LIN {X 0,Y 210.319,Z 902.747,A -85,B 0,C 180,E1 -29716.885,E2 -29716.885} C_VEL
LIN {X 0,Y 210.36,Z 916.958,A -85,B 0,C 180,E1 -29720.636,E2 -29720.636} C_VEL
LIN {X 0,Y 210.916,Z 920.236,A -85,B 0,C 180,E1 -29721.95,E2 -29721.95} C_VEL
LIN {X 0,Y 215.207,Z 930.512,A -85,B 0,C 180,E1 -29727.206,E2 -29727.206} C_VEL
LIN {X 0,Y 222.813,Z 941.87,A -85,B 0,C 180,E1 -29733.503,E2 -29733.503} C_VEL
LIN {X 0,Y 234.173,Z 953.754,A -85,B 0,C 180,E1 -29740.198,E2 -29740.198} C_VEL
LIN {X 0,Y 249.698,Z 966.285,A -85,B 0,C 180,E1 -29747.036,E2 -29747.036} C_VEL
LIN {X 0,Y 259.021,Z 973.419,A -85,B 0,C 180,E1 -29750.555,E2 -29750.555} C_VEL
LIN {X 0,Y 266.825,Z 979.349,A -85,B 0,C 180,E1 -29753.45,E2 -29753.45} C_VEL
LIN {X 0,Y 272.417,Z 983.731,A -85,B 0,C 180,E1 -29755.644,E2 -29755.644} C_VEL
LIN {X 0,Y 279.791,Z 989.154,A -85,B 0,C 180,E1 -29758.652,E2 -29758.652} C_VEL
LIN {X 0,Y 286.884,Z 994.471,A -85,B 0,C 180,E1 -29761.873,E2 -29761.873} C_VEL
LIN {X 0,Y 291.933,Z 998.076,A -85,B 0,C 180,E1 -29764.322,E2 -29764.322} C_VEL
LIN {X 0,Y 297.29,Z 1001.982,A -85,B 0,C 180,E1 -29767.214,E2 -29767.214} C_VEL
LIN {X 0,Y 301.306,Z 1004.65,A -85,B 0,C 180,E1 -29769.521,E2 -29769.521} C_VEL
LIN {X 0,Y 304.104,Z 1006.607,A -85,B 0,C 180,E1 -29771.355,E2 -29771.355} C_VEL
LIN {X 0,Y 307.657,Z 1009.394,A -85,B 0,C 180,E1 -29774.091,E2 -29774.091} C_VEL
LIN {X 0,Y 310.964,Z 1011.661,A -85,B 0,C 180,E1 -29776.938,E2 -29776.938} C_VEL
LIN {X 0,Y 314.05,Z 1013.321,A -85,B 0,C 180,E1 -29779.947,E2 -29779.947} C_VEL
LIN {X 0,Y 316.064,Z 1014.25,A -85,B 0,C 180,E1 -29782.333,E2 -29782.333} C_VEL
LIN {X 0,Y 317.605,Z 1014.95,A -85,B 0,C 180,E1 -29784.922,E2 -29784.922} C_VEL
LIN {X 0,Y 318.555,Z 1015.361,A -85,B 0,C 180,E1 -29787.471,E2 -29787.471} C_VEL
LIN {X 0,Y 318.776,Z 1015.511,A -85,B 0,C 180,E1 -29790,E2 -29790} C_VEL
LIN {X 0,Y 318.553,Z 1015.357,A -85,B 0,C 180,E1 -29792.529,E2 -29792.529} C_VEL
LIN {X 0,Y 317.534,Z 1014.981,A -85,B 0,C 180,E1 -29795.143,E2 -29795.143} C_VEL
LIN {X 0,Y 316.037,Z 1014.273,A -85,B 0,C 180,E1 -29797.667,E2 -29797.667} C_VEL
LIN {X 0,Y 313.796,Z 1013.227,A -85,B 0,C 180,E1 -29800.321,E2 -29800.321} C_VEL
LIN {X 0,Y 310.634,Z 1011.462,A -85,B 0,C 180,E1 -29803.382,E2 -29803.382} C_VEL
LIN {X 0,Y 307.344,Z 1009.146,A -85,B 0,C 180,E1 -29806.179,E2 -29806.179} C_VEL
LIN {X 0,Y 303.767,Z 1006.331,A -85,B 0,C 180,E1 -29808.899,E2 -29808.899} C_VEL
LIN {X 0,Y 300.741,Z 1004.289,A -85,B 0,C 180,E1 -29810.813,E2 -29810.813} C_VEL
LIN {X 0,Y 295.368,Z 1000.609,A -85,B 0,C 180,E1 -29813.859,E2 -29813.859} C_VEL
LIN {X 0,Y 290.463,Z 996.916,A -85,B 0,C 180,E1 -29816.462,E2 -29816.462} C_VEL
LIN {X 0,Y 285.122,Z 993.212,A -85,B 0,C 180,E1 -29818.951,E2 -29818.951} C_VEL
LIN {X 0,Y 278.129,Z 987.907,A -85,B 0,C 180,E1 -29822.048,E2 -29822.048} C_VEL
LIN {X 0,Y 270.582,Z 982.305,A -85,B 0,C 180,E1 -29825.098,E2 -29825.098} C_VEL
LIN {X 0,Y 263.436,Z 976.696,A -85,B 0,C 180,E1 -29827.849,E2 -29827.849} C_VEL
LIN {X 0,Y 253.442,Z 969.085,A -85,B 0,C 180,E1 -29831.522,E2 -29831.522} C_VEL
LIN {X 0,Y 239.695,Z 958.548,A -85,B 0,C 180,E1 -29837.138,E2 -29837.138} C_VEL
LIN {X 0,Y 225.348,Z 945.049,A -85,B 0,C 180,E1 -29844.763,E2 -29844.763} C_VEL
LIN {X 0,Y 217.144,Z 933.823,A -85,B 0,C 180,E1 -29850.957,E2 -29850.957} C_VEL
LIN {X 0,Y 212.466,Z 924.491,A -85,B 0,C 180,E1 -29855.923,E2 -29855.923} C_VEL
LIN {X 0,Y 209.033,Z 913.185,A -85,B 0,C 180,E1 -29861.437,E2 -29861.437} C_VEL
LIN {X 0,Y 207.187,Z 900.869,A -85,B 0,C 180,E1 -29866.932,E2 -29866.932} C_VEL
LIN {X 0,Y 206.615,Z 891.892,A -85,B 0,C 180,E1 -29870.748,E2 -29870.748} C_VEL
LIN {X 0,Y 206.248,Z 887.985,A -85,B 0,C 180,E1 -29872.997,E2 -29872.997} C_VEL
LIN {X 0,Y 205.868,Z 884.919,A -85,B 0,C 180,E1 -29875.595,E2 -29875.595} C_VEL
LIN {X 0,Y 205.707,Z 883.432,A -85,B 0,C 180,E1 -29877.553,E2 -29877.553} C_VEL
LIN {X 0,Y 205.644,Z 882.867,A -85,B 0,C 180,E1 -29879.359,E2 -29879.359} C_VEL
LIN {X 0,Y 202.968,Z 897.04,A -85,B 0,C 180,E1 -29879.559,E2 -29879.559} C_VEL
LIN {X 0,Y 199.768,Z 909.589,A -85,B 0,C 180,E1 -29879.721,E2 -29879.721} C_VEL
LIN {X 0,Y 196.126,Z 921.044,A -85,B 0,C 180,E1 -29879.878,E2 -29879.878} C_VEL
LIN {X 0,Y 191.11,Z 933.924,A -85,B 0,C 180,E1 -29880.105,E2 -29880.105} C_VEL
LIN {X 0,Y 185.363,Z 946.249,A -85,B 0,C 180,E1 -29880.387,E2 -29880.387} C_VEL
LIN {X 0,Y 178.348,Z 958.97,A -85,B 0,C 180,E1 -29880.8,E2 -29880.8} C_VEL
LIN {X 0,Y 171.342,Z 969.953,A -85,B 0,C 180,E1 -29881.224,E2 -29881.224} C_VEL
LIN {X 0,Y 163.472,Z 980.735,A -85,B 0,C 180,E1 -29881.747,E2 -29881.747} C_VEL
LIN {X 0,Y 154.751,Z 991.222,A -85,B 0,C 180,E1 -29882.433,E2 -29882.433} C_VEL
LIN {X 0,Y 146.063,Z 1000.482,A -85,B 0,C 180,E1 -29883.257,E2 -29883.257} C_VEL
LIN {X 0,Y 135.659,Z 1010.198,A -85,B 0,C 180,E1 -29884.256,E2 -29884.256} C_VEL
LIN {X 0,Y 125.327,Z 1018.712,A -85,B 0,C 180,E1 -29885.529,E2 -29885.529} C_VEL
LIN {X 0,Y 113.37,Z 1027.307,A -85,B 0,C 180,E1 -29887.326,E2 -29887.326} C_VEL
LIN {X 0,Y 103.236,Z 1033.736,A -85,B 0,C 180,E1 -29889.215,E2 -29889.215} C_VEL
LIN {X 0,Y 89.923,Z 1040.997,A -85,B 0,C 180,E1 -29892.335,E2 -29892.335} C_VEL
LIN {X 0,Y 80.172,Z 1045.652,A -85,B 0,C 180,E1 -29895.365,E2 -29895.365} C_VEL
LIN {X 0,Y 67.643,Z 1050.762,A -85,B 0,C 180,E1 -29900.762,E2 -29900.762} C_VEL
LIN {X 0,Y 55.947,Z 1054.78,A -85,B 0,C 180,E1 -29908.441,E2 -29908.441} C_VEL
LIN {X 0,Y 49.911,Z 1056.686,A -85,B 0,C 180,E1 -29914.283,E2 -29914.283} C_VEL
LIN {X 0,Y 41.398,Z 1058.964,A -85,B 0,C 180,E1 -29927.23,E2 -29927.23} C_VEL
LIN {X 0,Y 35.44,Z 1060.469,A -85,B 0,C 180,E1 -29946.634,E2 -29946.634} C_VEL
LIN {X 0,Y 34.109,Z 1060.992,A -85,B 0,C 180,E1 -29970,E2 -29970} C_VEL
LIN {X 0,Y 35.44,Z 1060.469,A -85,B 0,C 180,E1 -29993.366,E2 -29993.366} C_VEL
LIN {X 0,Y 41.398,Z 1058.964,A -85,B 0,C 180,E1 -30012.769,E2 -30012.769} C_VEL
LIN {X 0,Y 50.596,Z 1056.467,A -85,B 0,C 180,E1 -30026.449,E2 -30026.449} C_VEL
LIN {X 0,Y 64.625,Z 1051.854,A -85,B 0,C 180,E1 -30037.571,E2 -30037.571} C_VEL
LIN {X 0,Y 73.824,Z 1048.354,A -85,B 0,C 180,E1 -30042.169,E2 -30042.169} C_VEL
LIN {X 0,Y 86.648,Z 1042.62,A -85,B 0,C 180,E1 -30046.729,E2 -30046.729} C_VEL
LIN {X 0,Y 96.543,Z 1037.558,A -85,B 0,C 180,E1 -30049.335,E2 -30049.335} C_VEL
LIN {X 0,Y 109.975,Z 1029.527,A -85,B 0,C 180,E1 -30052.101,E2 -30052.101} C_VEL
LIN {X 0,Y 120.187,Z 1022.549,A -85,B 0,C 180,E1 -30053.749,E2 -30053.749} C_VEL
LIN {X 0,Y 130.479,Z 1014.587,A -85,B 0,C 180,E1 -30055.161,E2 -30055.161} C_VEL
LIN {X 0,Y 140.855,Z 1005.489,A -85,B 0,C 180,E1 -30056.268,E2 -30056.268} C_VEL
LIN {X 0,Y 150.25,Z 996.139,A -85,B 0,C 180,E1 -30057.21,E2 -30057.21} C_VEL
LIN {X 0,Y 159.981,Z 985.081,A -85,B 0,C 180,E1 -30057.989,E2 -30057.989} C_VEL
LIN {X 0,Y 168.717,Z 973.688,A -85,B 0,C 180,E1 -30058.615,E2 -30058.615} C_VEL
LIN {X 0,Y 176.596,Z 961.843,A -85,B 0,C 180,E1 -30059.088,E2 -30059.088} C_VEL
LIN {X 0,Y 182.731,Z 951.27,A -85,B 0,C 180,E1 -30059.473,E2 -30059.473} C_VEL
LIN {X 0,Y 188.873,Z 938.963,A -85,B 0,C 180,E1 -30059.807,E2 -30059.807} C_VEL
LIN {X 0,Y 194.039,Z 926.721,A -85,B 0,C 180,E1 -30060.042,E2 -30060.042} C_VEL
LIN {X 0,Y 198.913,Z 912.491,A -85,B 0,C 180,E1 -30060.258,E2 -30060.258} C_VEL
LIN {X 0,Y 202.152,Z 900.671,A -85,B 0,C 180,E1 -30060.396,E2 -30060.396} C_VEL
LIN {X 0,Y 204.983,Z 886.82,A -85,B 0,C 180,E1 -30060.57,E2 -30060.57} C_VEL
LIN {X 0,Y 205.603,Z 882.866,A -85,B 0,C 180,E1 -30060.66,E2 -30060.66} C_VEL
LIN {X 0,Y 205.7,Z 883.716,A -85,B 0,C 180,E1 -30062.998,E2 -30062.998} C_VEL
LIN {X 0,Y 205.985,Z 886.302,A -85,B 0,C 180,E1 -30065.69,E2 -30065.69} C_VEL
LIN {X 0,Y 206.423,Z 889.468,A -85,B 0,C 180,E1 -30067.95,E2 -30067.95} C_VEL
LIN {X 0,Y 206.719,Z 894.294,A -85,B 0,C 180,E1 -30070.334,E2 -30070.334} C_VEL
LIN {X 0,Y 207.984,Z 907.885,A -85,B 0,C 180,E1 -30076.124,E2 -30076.124} C_VEL
LIN {X 0,Y 210.642,Z 919.417,A -85,B 0,C 180,E1 -30081.531,E2 -30081.531} C_VEL
LIN {X 0,Y 210.916,Z 920.236,A -85,B 0,C 180,E1 -30081.95,E2 -30081.95} C_VEL
LIN {X 0,Y 211.624,Z 923.466,A -85,B 0,C 180,E1 -30083.276,E2 -30083.276} C_VEL
LIN {X 0,Y 212.413,Z 936.537,A -85,B 0,C 180,E1 -30087.282,E2 -30087.282} C_VEL
LIN {X 0,Y 213.319,Z 939.574,A -85,B 0,C 180,E1 -30088.616,E2 -30088.616} C_VEL
LIN {X 0,Y 222.269,Z 951.95,A -85,B 0,C 180,E1 -30095.799,E2 -30095.799} C_VEL
LIN {X 0,Y 237.602,Z 965.858,A -85,B 0,C 180,E1 -30104.034,E2 -30104.034} C_VEL
LIN {X 0,Y 250.262,Z 975.458,A -85,B 0,C 180,E1 -30109.307,E2 -30109.307} C_VEL
LIN {X 0,Y 260.2,Z 982.969,A -85,B 0,C 180,E1 -30113.048,E2 -30113.048} C_VEL
LIN {X 0,Y 267.131,Z 988.429,A -85,B 0,C 180,E1 -30115.757,E2 -30115.757} C_VEL
LIN {X 0,Y 273.023,Z 992.727,A -85,B 0,C 180,E1 -30118.152,E2 -30118.152} C_VEL
LIN {X 0,Y 280.748,Z 998.56,A -85,B 0,C 180,E1 -30121.6,E2 -30121.6} C_VEL
LIN {X 0,Y 285.146,Z 1001.663,A -85,B 0,C 180,E1 -30123.664,E2 -30123.664} C_VEL
LIN {X 0,Y 290.82,Z 1005.864,A -85,B 0,C 180,E1 -30126.679,E2 -30126.679} C_VEL
LIN {X 0,Y 295.051,Z 1008.723,A -85,B 0,C 180,E1 -30129.066,E2 -30129.066} C_VEL
LIN {X 0,Y 297.749,Z 1010.559,A -85,B 0,C 180,E1 -30130.758,E2 -30130.758} C_VEL
LIN {X 0,Y 301.06,Z 1013.064,A -85,B 0,C 180,E1 -30133.156,E2 -30133.156} C_VEL
LIN {X 0,Y 304.345,Z 1015.479,A -85,B 0,C 180,E1 -30135.897,E2 -30135.897} C_VEL
LIN {X 0,Y 307.762,Z 1017.533,A -85,B 0,C 180,E1 -30139.09,E2 -30139.09} C_VEL
LIN {X 0,Y 309.448,Z 1018.369,A -85,B 0,C 180,E1 -30140.853,E2 -30140.853} C_VEL
LIN {X 0,Y 311.43,Z 1019.222,A -85,B 0,C 180,E1 -30143.521,E2 -30143.521} C_VEL
LIN {X 0,Y 312.73,Z 1019.823,A -85,B 0,C 180,E1 -30146.134,E2 -30146.134} C_VEL
LIN {X 0,Y 313.157,Z 1019.993,A -85,B 0,C 180,E1 -30147.427,E2 -30147.427} C_VEL
LIN {X 0,Y 313.416,Z 1020.13,A -85,B 0,C 180,E1 -30150,E2 -30150} C_VEL
LIN {X 0,Y 313.152,Z 1019.992,A -85,B 0,C 180,E1 -30152.573,E2 -30152.573} C_VEL
LIN {X 0,Y 312.114,Z 1019.591,A -85,B 0,C 180,E1 -30155.167,E2 -30155.167} C_VEL
LIN {X 0,Y 310.513,Z 1018.854,A -85,B 0,C 180,E1 -30157.805,E2 -30157.805} C_VEL
LIN {X 0,Y 308.191,Z 1017.749,A -85,B 0,C 180,E1 -30160.511,E2 -30160.511} C_VEL
LIN {X 0,Y 305.255,Z 1016.052,A -85,B 0,C 180,E1 -30163.31,E2 -30163.31} C_VEL
LIN {X 0,Y 301.835,Z 1013.667,A -85,B 0,C 180,E1 -30166.225,E2 -30166.225} C_VEL
LIN {X 0,Y 299.93,Z 1012.106,A -85,B 0,C 180,E1 -30167.735,E2 -30167.735} C_VEL
LIN {X 0,Y 297.668,Z 1010.499,A -85,B 0,C 180,E1 -30169.301,E2 -30169.301} C_VEL
LIN {X 0,Y 294.302,Z 1008.221,A -85,B 0,C 180,E1 -30171.359,E2 -30171.359} C_VEL
LIN {X 0,Y 288.802,Z 1004.324,A -85,B 0,C 180,E1 -30174.436,E2 -30174.436} C_VEL
LIN {X 0,Y 283.861,Z 1000.701,A -85,B 0,C 180,E1 -30176.963,E2 -30176.963} C_VEL
LIN {X 0,Y 278.805,Z 997.204,A -85,B 0,C 180,E1 -30179.275,E2 -30179.275} C_VEL
LIN {X 0,Y 273.007,Z 992.71,A -85,B 0,C 180,E1 -30181.842,E2 -30181.842} C_VEL
LIN {X 0,Y 267.168,Z 988.423,A -85,B 0,C 180,E1 -30184.212,E2 -30184.212} C_VEL
LIN {X 0,Y 260.219,Z 983.003,A -85,B 0,C 180,E1 -30186.928,E2 -30186.928} C_VEL
LIN {X 0,Y 250.27,Z 975.447,A -85,B 0,C 180,E1 -30190.695,E2 -30190.695} C_VEL
LIN {X 0,Y 235.873,Z 964.545,A -85,B 0,C 180,E1 -30196.742,E2 -30196.742} C_VEL
LIN {X 0,Y 220.949,Z 950.497,A -85,B 0,C 180,E1 -30205.073,E2 -30205.073} C_VEL
LIN {X 0,Y 213.252,Z 939.448,A -85,B 0,C 180,E1 -30211.455,E2 -30211.455} C_VEL
LIN {X 0,Y 208.566,Z 928.974,A -85,B 0,C 180,E1 -30217.201,E2 -30217.201} C_VEL
LIN {X 0,Y 205.852,Z 917.557,A -85,B 0,C 180,E1 -30222.925,E2 -30222.925} C_VEL
LIN {X 0,Y 204.846,Z 904.198,A -85,B 0,C 180,E1 -30228.936,E2 -30228.936} C_VEL
LIN {X 0,Y 204.751,Z 897.765,A -85,B 0,C 180,E1 -30231.75,E2 -30231.75} C_VEL
LIN {X 0,Y 204.648,Z 894.053,A -85,B 0,C 180,E1 -30233.963,E2 -30233.963} C_VEL
LIN {X 0,Y 204.566,Z 891.702,A -85,B 0,C 180,E1 -30236.061,E2 -30236.061} C_VEL
LIN {X 0,Y 204.548,Z 890.533,A -85,B 0,C 180,E1 -30237.44,E2 -30237.44} C_VEL
LIN {X 0,Y 200.464,Z 907.587,A -85,B 0,C 180,E1 -30237.662,E2 -30237.662} C_VEL
LIN {X 0,Y 196.214,Z 921,A -85,B 0,C 180,E1 -30237.805,E2 -30237.805} C_VEL
LIN {X 0,Y 191.235,Z 933.711,A -85,B 0,C 180,E1 -30237.98,E2 -30237.98} C_VEL
LIN {X 0,Y 185.451,Z 946.049,A -85,B 0,C 180,E1 -30238.185,E2 -30238.185} C_VEL
LIN {X 0,Y 178.391,Z 958.769,A -85,B 0,C 180,E1 -30238.514,E2 -30238.514} C_VEL
LIN {X 0,Y 171.338,Z 969.752,A -85,B 0,C 180,E1 -30238.834,E2 -30238.834} C_VEL
LIN {X 0,Y 163.411,Z 980.531,A -85,B 0,C 180,E1 -30239.233,E2 -30239.233} C_VEL
LIN {X 0,Y 154.613,Z 991.02,A -85,B 0,C 180,E1 -30239.78,E2 -30239.78} C_VEL
LIN {X 0,Y 145.831,Z 1000.279,A -85,B 0,C 180,E1 -30240.447,E2 -30240.447} C_VEL
LIN {X 0,Y 135.317,Z 1009.995,A -85,B 0,C 180,E1 -30241.234,E2 -30241.234} C_VEL
LIN {X 0,Y 124.839,Z 1018.508,A -85,B 0,C 180,E1 -30242.244,E2 -30242.244} C_VEL
LIN {X 0,Y 112.677,Z 1027.1,A -85,B 0,C 180,E1 -30243.674,E2 -30243.674} C_VEL
LIN {X 0,Y 102.331,Z 1033.529,A -85,B 0,C 180,E1 -30245.239,E2 -30245.239} C_VEL
LIN {X 0,Y 88.664,Z 1040.788,A -85,B 0,C 180,E1 -30247.783,E2 -30247.783} C_VEL
LIN {X 0,Y 78.416,Z 1045.505,A -85,B 0,C 180,E1 -30250.327,E2 -30250.327} C_VEL
LIN {X 0,Y 65.438,Z 1050.554,A -85,B 0,C 180,E1 -30254.856,E2 -30254.856} C_VEL
LIN {X 0,Y 52.892,Z 1054.571,A -85,B 0,C 180,E1 -30261.55,E2 -30261.55} C_VEL
LIN {X 0,Y 45.411,Z 1056.683,A -85,B 0,C 180,E1 -30267.667,E2 -30267.667} C_VEL
LIN {X 0,Y 36.459,Z 1058.757,A -85,B 0,C 180,E1 -30279.553,E2 -30279.553} C_VEL
LIN {X 0,Y 29.002,Z 1060.261,A -85,B 0,C 180,E1 -30301.011,E2 -30301.011} C_VEL
LIN {X 0,Y 26.998,Z 1060.786,A -85,B 0,C 180,E1 -30330,E2 -30330} C_VEL
LIN {X 0,Y 29.002,Z 1060.261,A -85,B 0,C 180,E1 -30358.989,E2 -30358.989} C_VEL
LIN {X 0,Y 36.461,Z 1058.757,A -85,B 0,C 180,E1 -30380.444,E2 -30380.444} C_VEL
LIN {X 0,Y 47,Z 1056.259,A -85,B 0,C 180,E1 -30393.789,E2 -30393.789} C_VEL
LIN {X 0,Y 62.231,Z 1051.646,A -85,B 0,C 180,E1 -30403.723,E2 -30403.723} C_VEL
LIN {X 0,Y 71.943,Z 1048.145,A -85,B 0,C 180,E1 -30407.648,E2 -30407.648} C_VEL
LIN {X 0,Y 85.282,Z 1042.411,A -85,B 0,C 180,E1 -30411.448,E2 -30411.448} C_VEL
LIN {X 0,Y 95.472,Z 1037.35,A -85,B 0,C 180,E1 -30413.592,E2 -30413.592} C_VEL
LIN {X 0,Y 109.219,Z 1029.322,A -85,B 0,C 180,E1 -30415.835,E2 -30415.835} C_VEL
LIN {X 0,Y 119.617,Z 1022.343,A -85,B 0,C 180,E1 -30417.182,E2 -30417.182} C_VEL
LIN {X 0,Y 130.071,Z 1014.383,A -85,B 0,C 180,E1 -30418.318,E2 -30418.318} C_VEL
LIN {X 0,Y 140.571,Z 1005.286,A -85,B 0,C 180,E1 -30419.178,E2 -30419.178} C_VEL
LIN {X 0,Y 150.894,Z 995.045,A -85,B 0,C 180,E1 -30419.999,E2 -30419.999} C_VEL
LIN {X 0,Y 159.89,Z 984.877,A -85,B 0,C 180,E1 -30420.555,E2 -30420.555} C_VEL
LIN {X 0,Y 168.695,Z 973.487,A -85,B 0,C 180,E1 -30421.04,E2 -30421.04} C_VEL
LIN {X 0,Y 176.626,Z 961.642,A -85,B 0,C 180,E1 -30421.4,E2 -30421.4} C_VEL
LIN {X 0,Y 182.804,Z 951.071,A -85,B 0,C 180,E1 -30421.702,E2 -30421.702} C_VEL
LIN {X 0,Y 188.984,Z 938.764,A -85,B 0,C 180,E1 -30421.966,E2 -30421.966} C_VEL
LIN {X 0,Y 194.63,Z 925.293,A -85,B 0,C 180,E1 -30422.157,E2 -30422.157} C_VEL
LIN {X 0,Y 199.099,Z 912.2,A -85,B 0,C 180,E1 -30422.299,E2 -30422.299} C_VEL
LIN {X 0,Y 202.327,Z 900.481,A -85,B 0,C 180,E1 -30422.415,E2 -30422.415} C_VEL
LIN {X 0,Y 204.546,Z 890.534,A -85,B 0,C 180,E1 -30422.547,E2 -30422.547} C_VEL
LIN {X 0,Y 204.612,Z 893.203,A -85,B 0,C 180,E1 -30425.357,E2 -30425.357} C_VEL
LIN {X 0,Y 204.706,Z 896.076,A -85,B 0,C 180,E1 -30427.335,E2 -30427.335} C_VEL
LIN {X 0,Y 204.806,Z 900.672,A -85,B 0,C 180,E1 -30429.578,E2 -30429.578} C_VEL
LIN {X 0,Y 205.536,Z 915.012,A -85,B 0,C 180,E1 -30435.875,E2 -30435.875} C_VEL
LIN {X 0,Y 207.672,Z 926.02,A -85,B 0,C 180,E1 -30441.273,E2 -30441.273} C_VEL
LIN {X 0,Y 211.409,Z 936.153,A -85,B 0,C 180,E1 -30446.665,E2 -30446.665} C_VEL
LIN {X 0,Y 213.319,Z 939.574,A -85,B 0,C 180,E1 -30448.616,E2 -30448.616} C_VEL
LIN {X 0,Y 214.347,Z 942.536,A -85,B 0,C 180,E1 -30449.963,E2 -30449.963} C_VEL
LIN {X 0,Y 216.225,Z 954.474,A -85,B 0,C 180,E1 -30454.145,E2 -30454.145} C_VEL
LIN {X 0,Y 217.597,Z 957.177,A -85,B 0,C 180,E1 -30455.478,E2 -30455.478} C_VEL
LIN {X 0,Y 230.366,Z 969.155,A -85,B 0,C 180,E1 -30462.931,E2 -30462.931} C_VEL
LIN {X 0,Y 243.238,Z 978.893,A -85,B 0,C 180,E1 -30468.696,E2 -30468.696} C_VEL
LIN {X 0,Y 254.634,Z 987.392,A -85,B 0,C 180,E1 -30473.168,E2 -30473.168} C_VEL
LIN {X 0,Y 260.627,Z 992.11,A -85,B 0,C 180,E1 -30475.51,E2 -30475.51} C_VEL
LIN {X 0,Y 267.549,Z 997.165,A -85,B 0,C 180,E1 -30478.308,E2 -30478.308} C_VEL
LIN {X 0,Y 273.403,Z 1001.729,A -85,B 0,C 180,E1 -30480.924,E2 -30480.924} C_VEL
LIN {X 0,Y 278.901,Z 1005.585,A -85,B 0,C 180,E1 -30483.449,E2 -30483.449} C_VEL
LIN {X 0,Y 284.194,Z 1009.505,A -85,B 0,C 180,E1 -30486.203,E2 -30486.203} C_VEL
LIN {X 0,Y 288.419,Z 1012.428,A -85,B 0,C 180,E1 -30488.562,E2 -30488.562} C_VEL
LIN {X 0,Y 291.253,Z 1014.333,A -85,B 0,C 180,E1 -30490.256,E2 -30490.256} C_VEL
LIN {X 0,Y 294.633,Z 1016.738,A -85,B 0,C 180,E1 -30492.578,E2 -30492.578} C_VEL
LIN {X 0,Y 297.94,Z 1019.258,A -85,B 0,C 180,E1 -30495.267,E2 -30495.267} C_VEL
LIN {X 0,Y 301.367,Z 1021.447,A -85,B 0,C 180,E1 -30498.362,E2 -30498.362} C_VEL
LIN {X 0,Y 303.646,Z 1022.632,A -85,B 0,C 180,E1 -30500.676,E2 -30500.676} C_VEL
LIN {X 0,Y 305.73,Z 1023.531,A -85,B 0,C 180,E1 -30503.4,E2 -30503.4} C_VEL
LIN {X 0,Y 307.118,Z 1024.17,A -85,B 0,C 180,E1 -30506.064,E2 -30506.064} C_VEL
LIN {X 0,Y 307.561,Z 1024.36,A -85,B 0,C 180,E1 -30507.381,E2 -30507.381} C_VEL
LIN {X 0,Y 307.836,Z 1024.509,A -85,B 0,C 180,E1 -30510,E2 -30510} C_VEL
LIN {X 0,Y 307.556,Z 1024.358,A -85,B 0,C 180,E1 -30512.619,E2 -30512.619} C_VEL
LIN {X 0,Y 306.446,Z 1023.932,A -85,B 0,C 180,E1 -30515.263,E2 -30515.263} C_VEL
LIN {X 0,Y 304.758,Z 1023.131,A -85,B 0,C 180,E1 -30517.953,E2 -30517.953} C_VEL
LIN {X 0,Y 302.323,Z 1022.004,A -85,B 0,C 180,E1 -30520.718,E2 -30520.718} C_VEL
LIN {X 0,Y 299.264,Z 1020.174,A -85,B 0,C 180,E1 -30523.582,E2 -30523.582} C_VEL
LIN {X 0,Y 295.762,Z 1017.62,A -85,B 0,C 180,E1 -30526.567,E2 -30526.567} C_VEL
LIN {X 0,Y 293.679,Z 1016.019,A -85,B 0,C 180,E1 -30528.125,E2 -30528.125} C_VEL
LIN {X 0,Y 291.234,Z 1014.319,A -85,B 0,C 180,E1 -30529.758,E2 -30529.758} C_VEL
LIN {X 0,Y 287.715,Z 1011.923,A -85,B 0,C 180,E1 -30531.842,E2 -30531.842} C_VEL
LIN {X 0,Y 284.213,Z 1009.472,A -85,B 0,C 180,E1 -30533.806,E2 -30533.806} C_VEL
LIN {X 0,Y 278.924,Z 1005.545,A -85,B 0,C 180,E1 -30536.561,E2 -30536.561} C_VEL
LIN {X 0,Y 272.954,Z 1001.377,A -85,B 0,C 180,E1 -30539.288,E2 -30539.288} C_VEL
LIN {X 0,Y 267.482,Z 997.137,A -85,B 0,C 180,E1 -30541.7,E2 -30541.7} C_VEL
LIN {X 0,Y 260.581,Z 991.997,A -85,B 0,C 180,E1 -30544.497,E2 -30544.497} C_VEL
LIN {X 0,Y 252.706,Z 985.889,A -85,B 0,C 180,E1 -30547.572,E2 -30547.572} C_VEL
LIN {X 0,Y 241.442,Z 977.648,A -85,B 0,C 180,E1 -30552.027,E2 -30552.027} C_VEL
LIN {X 0,Y 229.277,Z 968.329,A -85,B 0,C 180,E1 -30557.596,E2 -30557.596} C_VEL
LIN {X 0,Y 216.427,Z 955.822,A -85,B 0,C 180,E1 -30565.371,E2 -30565.371} C_VEL
LIN {X 0,Y 209.16,Z 944.954,A -85,B 0,C 180,E1 -30571.94,E2 -30571.94} C_VEL
LIN {X 0,Y 205.516,Z 936.48,A -85,B 0,C 180,E1 -30576.844,E2 -30576.844} C_VEL
LIN {X 0,Y 203.125,Z 925.371,A -85,B 0,C 180,E1 -30582.689,E2 -30582.689} C_VEL
LIN {X 0,Y 202.471,Z 913.857,A -85,B 0,C 180,E1 -30588.17,E2 -30588.17} C_VEL
LIN {X 0,Y 202.912,Z 903.788,A -85,B 0,C 180,E1 -30592.663,E2 -30592.663} C_VEL
LIN {X 0,Y 202.969,Z 900.443,A -85,B 0,C 180,E1 -30594.677,E2 -30594.677} C_VEL
LIN {X 0,Y 202.96,Z 899.417,A -85,B 0,C 180,E1 -30595.531,E2 -30595.531} C_VEL
LIN {X 0,Y 199.77,Z 911.123,A -85,B 0,C 180,E1 -30595.66,E2 -30595.66} C_VEL
LIN {X 0,Y 195.372,Z 924.158,A -85,B 0,C 180,E1 -30595.761,E2 -30595.761} C_VEL
LIN {X 0,Y 190.243,Z 936.587,A -85,B 0,C 180,E1 -30595.878,E2 -30595.878} C_VEL
LIN {X 0,Y 184.925,Z 947.525,A -85,B 0,C 180,E1 -30596.025,E2 -30596.025} C_VEL
LIN {X 0,Y 178.717,Z 958.568,A -85,B 0,C 180,E1 -30596.232,E2 -30596.232} C_VEL
LIN {X 0,Y 171.631,Z 969.552,A -85,B 0,C 180,E1 -30596.455,E2 -30596.455} C_VEL
LIN {X 0,Y 162.777,Z 981.414,A -85,B 0,C 180,E1 -30596.769,E2 -30596.769} C_VEL
LIN {X 0,Y 154.806,Z 990.817,A -85,B 0,C 180,E1 -30597.133,E2 -30597.133} C_VEL
LIN {X 0,Y 145.952,Z 1000.074,A -85,B 0,C 180,E1 -30597.628,E2 -30597.628} C_VEL
LIN {X 0,Y 135.352,Z 1009.792,A -85,B 0,C 180,E1 -30598.203,E2 -30598.203} C_VEL
LIN {X 0,Y 124.765,Z 1018.303,A -85,B 0,C 180,E1 -30598.946,E2 -30598.946} C_VEL
LIN {X 0,Y 112.445,Z 1026.895,A -85,B 0,C 180,E1 -30600.011,E2 -30600.011} C_VEL
LIN {X 0,Y 101.925,Z 1033.323,A -85,B 0,C 180,E1 -30601.196,E2 -30601.196} C_VEL
LIN {X 0,Y 87.978,Z 1040.583,A -85,B 0,C 180,E1 -30603.116,E2 -30603.116} C_VEL
LIN {X 0,Y 76.44,Z 1045.693,A -85,B 0,C 180,E1 -30605.277,E2 -30605.277} C_VEL
LIN {X 0,Y 63.967,Z 1050.346,A -85,B 0,C 180,E1 -30608.587,E2 -30608.587} C_VEL
LIN {X 0,Y 50.694,Z 1054.363,A -85,B 0,C 180,E1 -30613.969,E2 -30613.969} C_VEL
LIN {X 0,Y 38.128,Z 1057.346,A -85,B 0,C 180,E1 -30622.836,E2 -30622.836} C_VEL
LIN {X 0,Y 32.351,Z 1058.548,A -85,B 0,C 180,E1 -30629.664,E2 -30629.664} C_VEL
LIN {X 0,Y 23.005,Z 1060.054,A -85,B 0,C 180,E1 -30652.34,E2 -30652.34} C_VEL
LIN {X 0,Y 19.878,Z 1060.58,A -85,B 0,C 180,E1 -30690,E2 -30690} C_VEL
LIN {X 0,Y 23.005,Z 1060.054,A -85,B 0,C 180,E1 -30727.66,E2 -30727.66} C_VEL
LIN {X 0,Y 32.355,Z 1058.548,A -85,B 0,C 180,E1 -30750.323,E2 -30750.323} C_VEL
LIN {X 0,Y 44.286,Z 1056.05,A -85,B 0,C 180,E1 -30762.205,E2 -30762.205} C_VEL
LIN {X 0,Y 60.608,Z 1051.438,A -85,B 0,C 180,E1 -30770.27,E2 -30770.27} C_VEL
LIN {X 0,Y 70.752,Z 1047.938,A -85,B 0,C 180,E1 -30773.363,E2 -30773.363} C_VEL
LIN {X 0,Y 84.511,Z 1042.206,A -85,B 0,C 180,E1 -30776.286,E2 -30776.286} C_VEL
LIN {X 0,Y 94.938,Z 1037.144,A -85,B 0,C 180,E1 -30777.911,E2 -30777.911} C_VEL
LIN {X 0,Y 108.934,Z 1029.118,A -85,B 0,C 180,E1 -30779.605,E2 -30779.605} C_VEL
LIN {X 0,Y 119.48,Z 1022.139,A -85,B 0,C 180,E1 -30780.62,E2 -30780.62} C_VEL
LIN {X 0,Y 130.058,Z 1014.18,A -85,B 0,C 180,E1 -30781.476,E2 -30781.476} C_VEL
LIN {X 0,Y 140.651,Z 1005.081,A -85,B 0,C 180,E1 -30782.105,E2 -30782.105} C_VEL
LIN {X 0,Y 150.414,Z 995.541,A -85,B 0,C 180,E1 -30782.677,E2 -30782.677} C_VEL
LIN {X 0,Y 160.118,Z 984.674,A -85,B 0,C 180,E1 -30783.108,E2 -30783.108} C_VEL
LIN {X 0,Y 168.975,Z 973.286,A -85,B 0,C 180,E1 -30783.46,E2 -30783.46} C_VEL
LIN {X 0,Y 176.944,Z 961.44,A -85,B 0,C 180,E1 -30783.71,E2 -30783.71} C_VEL
LIN {X 0,Y 183.153,Z 950.872,A -85,B 0,C 180,E1 -30783.926,E2 -30783.926} C_VEL
LIN {X 0,Y 189.362,Z 938.564,A -85,B 0,C 180,E1 -30784.121,E2 -30784.121} C_VEL
LIN {X 0,Y 194.798,Z 925.715,A -85,B 0,C 180,E1 -30784.238,E2 -30784.238} C_VEL
LIN {X 0,Y 199.509,Z 912.005,A -85,B 0,C 180,E1 -30784.335,E2 -30784.335} C_VEL
LIN {X 0,Y 202.818,Z 899.994,A -85,B 0,C 180,E1 -30784.422,E2 -30784.422} C_VEL
LIN {X 0,Y 202.95,Z 899.436,A -85,B 0,C 180,E1 -30784.449,E2 -30784.449} C_VEL
LIN {X 0,Y 202.961,Z 902.093,A -85,B 0,C 180,E1 -30786.399,E2 -30786.399} C_VEL
LIN {X 0,Y 202.737,Z 906.212,A -85,B 0,C 180,E1 -30788.472,E2 -30788.472} C_VEL
LIN {X 0,Y 202.581,Z 919.804,A -85,B 0,C 180,E1 -30794.567,E2 -30794.567} C_VEL
LIN {X 0,Y 204.05,Z 930.923,A -85,B 0,C 180,E1 -30800.146,E2 -30800.146} C_VEL
LIN {X 0,Y 207.518,Z 941.746,A -85,B 0,C 180,E1 -30806.12,E2 -30806.12} C_VEL
LIN {X 0,Y 214.151,Z 952.784,A -85,B 0,C 180,E1 -30812.785,E2 -30812.785} C_VEL
LIN {X 0,Y 217.597,Z 957.177,A -85,B 0,C 180,E1 -30815.478,E2 -30815.478} C_VEL
LIN {X 0,Y 219.18,Z 959.806,A -85,B 0,C 180,E1 -30816.805,E2 -30816.805} C_VEL
LIN {X 0,Y 222.356,Z 970.718,A -85,B 0,C 180,E1 -30821.023,E2 -30821.023} C_VEL
LIN {X 0,Y 224.174,Z 973.228,A -85,B 0,C 180,E1 -30822.313,E2 -30822.313} C_VEL
LIN {X 0,Y 238.097,Z 983.708,A -85,B 0,C 180,E1 -30828.889,E2 -30828.889} C_VEL
LIN {X 0,Y 250.333,Z 992.703,A -85,B 0,C 180,E1 -30833.875,E2 -30833.875} C_VEL
LIN {X 0,Y 258.896,Z 999.276,A -85,B 0,C 180,E1 -30837.3,E2 -30837.3} C_VEL
LIN {X 0,Y 264.592,Z 1003.463,A -85,B 0,C 180,E1 -30839.691,E2 -30839.691} C_VEL
LIN {X 0,Y 270.131,Z 1007.604,A -85,B 0,C 180,E1 -30842.198,E2 -30842.198} C_VEL
LIN {X 0,Y 275.626,Z 1011.504,A -85,B 0,C 180,E1 -30844.845,E2 -30844.845} C_VEL
LIN {X 0,Y 279.963,Z 1014.692,A -85,B 0,C 180,E1 -30847.168,E2 -30847.168} C_VEL
LIN {X 0,Y 284.552,Z 1017.852,A -85,B 0,C 180,E1 -30849.806,E2 -30849.806} C_VEL
LIN {X 0,Y 288.037,Z 1020.26,A -85,B 0,C 180,E1 -30852.096,E2 -30852.096} C_VEL
LIN {X 0,Y 291.263,Z 1022.728,A -85,B 0,C 180,E1 -30854.608,E2 -30854.608} C_VEL
LIN {X 0,Y 294.869,Z 1025.12,A -85,B 0,C 180,E1 -30857.74,E2 -30857.74} C_VEL
LIN {X 0,Y 297.594,Z 1026.59,A -85,B 0,C 180,E1 -30860.485,E2 -30860.485} C_VEL
LIN {X 0,Y 299.806,Z 1027.578,A -85,B 0,C 180,E1 -30863.269,E2 -30863.269} C_VEL
LIN {X 0,Y 301.3,Z 1028.259,A -85,B 0,C 180,E1 -30865.987,E2 -30865.987} C_VEL
LIN {X 0,Y 301.752,Z 1028.473,A -85,B 0,C 180,E1 -30867.33,E2 -30867.33} C_VEL
LIN {X 0,Y 302.058,Z 1028.627,A -85,B 0,C 180,E1 -30870,E2 -30870} C_VEL
LIN {X 0,Y 301.743,Z 1028.474,A -85,B 0,C 180,E1 -30872.67,E2 -30872.67} C_VEL
LIN {X 0,Y 300.582,Z 1027.998,A -85,B 0,C 180,E1 -30875.366,E2 -30875.366} C_VEL
LIN {X 0,Y 298.766,Z 1027.145,A -85,B 0,C 180,E1 -30878.114,E2 -30878.114} C_VEL
LIN {X 0,Y 296.233,Z 1025.937,A -85,B 0,C 180,E1 -30880.941,E2 -30880.941} C_VEL
LIN {X 0,Y 293.056,Z 1023.973,A -85,B 0,C 180,E1 -30883.875,E2 -30883.875} C_VEL
LIN {X 0,Y 289.408,Z 1021.258,A -85,B 0,C 180,E1 -30886.942,E2 -30886.942} C_VEL
LIN {X 0,Y 287.121,Z 1019.6,A -85,B 0,C 180,E1 -30888.554,E2 -30888.554} C_VEL
LIN {X 0,Y 283.054,Z 1016.798,A -85,B 0,C 180,E1 -30891.101,E2 -30891.101} C_VEL
LIN {X 0,Y 277.452,Z 1012.826,A -85,B 0,C 180,E1 -30894.233,E2 -30894.233} C_VEL
LIN {X 0,Y 272.028,Z 1008.881,A -85,B 0,C 180,E1 -30896.961,E2 -30896.961} C_VEL
LIN {X 0,Y 266.428,Z 1004.93,A -85,B 0,C 180,E1 -30899.485,E2 -30899.485} C_VEL
LIN {X 0,Y 260.836,Z 1000.576,A -85,B 0,C 180,E1 -30901.927,E2 -30901.927} C_VEL
LIN {X 0,Y 253.145,Z 994.84,A -85,B 0,C 180,E1 -30905.016,E2 -30905.016} C_VEL
LIN {X 0,Y 243.571,Z 987.722,A -85,B 0,C 180,E1 -30908.827,E2 -30908.827} C_VEL
LIN {X 0,Y 230.398,Z 978.08,A -85,B 0,C 180,E1 -30914.553,E2 -30914.553} C_VEL
LIN {X 0,Y 215.494,Z 965.204,A -85,B 0,C 180,E1 -30922.938,E2 -30922.938} C_VEL
LIN {X 0,Y 206.406,Z 953.18,A -85,B 0,C 180,E1 -30930.737,E2 -30930.737} C_VEL
LIN {X 0,Y 201.557,Z 941.119,A -85,B 0,C 180,E1 -30937.996,E2 -30937.996} C_VEL
LIN {X 0,Y 199.786,Z 928.716,A -85,B 0,C 180,E1 -30944.703,E2 -30944.703} C_VEL
LIN {X 0,Y 200.301,Z 914.658,A -85,B 0,C 180,E1 -30951.361,E2 -30951.361} C_VEL
LIN {X 0,Y 200.807,Z 909.691,A -85,B 0,C 180,E1 -30953.614,E2 -30953.614} C_VEL
LIN {X 0,Y 196.6,Z 922.411,A -85,B 0,C 180,E1 -30953.687,E2 -30953.687} C_VEL
LIN {X 0,Y 191.574,Z 934.851,A -85,B 0,C 180,E1 -30953.745,E2 -30953.745} C_VEL
LIN {X 0,Y 186.445,Z 945.652,A -85,B 0,C 180,E1 -30953.812,E2 -30953.812} C_VEL
LIN {X 0,Y 179.326,Z 958.366,A -85,B 0,C 180,E1 -30953.962,E2 -30953.962} C_VEL
LIN {X 0,Y 172.221,Z 969.351,A -85,B 0,C 180,E1 -30954.081,E2 -30954.081} C_VEL
LIN {X 0,Y 163.333,Z 981.211,A -85,B 0,C 180,E1 -30954.275,E2 -30954.275} C_VEL
LIN {X 0,Y 155.329,Z 990.615,A -85,B 0,C 180,E1 -30954.493,E2 -30954.493} C_VEL
LIN {X 0,Y 146.425,Z 999.87,A -85,B 0,C 180,E1 -30954.819,E2 -30954.819} C_VEL
LIN {X 0,Y 135.766,Z 1009.588,A -85,B 0,C 180,E1 -30955.176,E2 -30955.176} C_VEL
LIN {X 0,Y 125.104,Z 1018.098,A -85,B 0,C 180,E1 -30955.648,E2 -30955.648} C_VEL
LIN {X 0,Y 112.674,Z 1026.691,A -85,B 0,C 180,E1 -30956.349,E2 -30956.349} C_VEL
LIN {X 0,Y 102.03,Z 1033.117,A -85,B 0,C 180,E1 -30957.143,E2 -30957.143} C_VEL
LIN {X 0,Y 87.881,Z 1040.377,A -85,B 0,C 180,E1 -30958.414,E2 -30958.414} C_VEL
LIN {X 0,Y 75.229,Z 1045.828,A -85,B 0,C 180,E1 -30960.001,E2 -30960.001} C_VEL
LIN {X 0,Y 63.294,Z 1050.14,A -85,B 0,C 180,E1 -30962.121,E2 -30962.121} C_VEL
LIN {X 0,Y 49.451,Z 1054.157,A -85,B 0,C 180,E1 -30965.833,E2 -30965.833} C_VEL
LIN {X 0,Y 35.949,Z 1057.138,A -85,B 0,C 180,E1 -30972.184,E2 -30972.184} C_VEL
LIN {X 0,Y 29.458,Z 1058.341,A -85,B 0,C 180,E1 -30977.395,E2 -30977.395} C_VEL
LIN {X 0,Y 17.875,Z 1059.847,A -85,B 0,C 180,E1 -30998.154,E2 -30998.154} C_VEL
LIN {X 0,Y 12.751,Z 1060.374,A -85,B 0,C 180,E1 -31050,E2 -31050} C_VEL
LIN {X 0,Y 17.875,Z 1059.847,A -85,B 0,C 180,E1 -31101.845,E2 -31101.845} C_VEL
LIN {X 0,Y 29.462,Z 1058.341,A -85,B 0,C 180,E1 -31122.58,E2 -31122.58} C_VEL
LIN {X 0,Y 42.638,Z 1055.843,A -85,B 0,C 180,E1 -31131.474,E2 -31131.474} C_VEL
LIN {X 0,Y 59.812,Z 1051.232,A -85,B 0,C 180,E1 -31137.113,E2 -31137.113} C_VEL
LIN {X 0,Y 70.285,Z 1047.731,A -85,B 0,C 180,E1 -31139.207,E2 -31139.207} C_VEL
LIN {X 0,Y 84.351,Z 1042,A -85,B 0,C 180,E1 -31141.177,E2 -31141.177} C_VEL
LIN {X 0,Y 94.949,Z 1036.938,A -85,B 0,C 180,E1 -31142.261,E2 -31142.261} C_VEL
LIN {X 0,Y 108.757,Z 1029.141,A -85,B 0,C 180,E1 -31143.369,E2 -31143.369} C_VEL
LIN {X 0,Y 119.775,Z 1021.933,A -85,B 0,C 180,E1 -31144.07,E2 -31144.07} C_VEL
LIN {X 0,Y 130.44,Z 1013.976,A -85,B 0,C 180,E1 -31144.632,E2 -31144.632} C_VEL
LIN {X 0,Y 141.094,Z 1004.878,A -85,B 0,C 180,E1 -31145.006,E2 -31145.006} C_VEL
LIN {X 0,Y 150.218,Z 996.087,A -85,B 0,C 180,E1 -31145.368,E2 -31145.368} C_VEL
LIN {X 0,Y 160.664,Z 984.471,A -85,B 0,C 180,E1 -31145.652,E2 -31145.652} C_VEL
LIN {X 0,Y 169.556,Z 973.085,A -85,B 0,C 180,E1 -31145.868,E2 -31145.868} C_VEL
LIN {X 0,Y 177.551,Z 961.238,A -85,B 0,C 180,E1 -31146.015,E2 -31146.015} C_VEL
LIN {X 0,Y 184.667,Z 948.999,A -85,B 0,C 180,E1 -31146.158,E2 -31146.158} C_VEL
LIN {X 0,Y 190.005,Z 938.365,A -85,B 0,C 180,E1 -31146.26,E2 -31146.26} C_VEL
LIN {X 0,Y 195.587,Z 925.152,A -85,B 0,C 180,E1 -31146.317,E2 -31146.317} C_VEL
LIN {X 0,Y 200.254,Z 911.533,A -85,B 0,C 180,E1 -31146.369,E2 -31146.369} C_VEL
LIN {X 0,Y 200.796,Z 909.774,A -85,B 0,C 180,E1 -31146.424,E2 -31146.424} C_VEL
LIN {X 0,Y 199.711,Z 922.383,A -85,B 0,C 180,E1 -31152.189,E2 -31152.189} C_VEL
LIN {X 0,Y 200.233,Z 934.682,A -85,B 0,C 180,E1 -31158.414,E2 -31158.414} C_VEL
LIN {X 0,Y 202.822,Z 945.568,A -85,B 0,C 180,E1 -31164.57,E2 -31164.57} C_VEL
LIN {X 0,Y 208.548,Z 956.625,A -85,B 0,C 180,E1 -31171.489,E2 -31171.489} C_VEL
LIN {X 0,Y 218.26,Z 968.016,A -85,B 0,C 180,E1 -31178.895,E2 -31178.895} C_VEL
LIN {X 0,Y 224.174,Z 973.228,A -85,B 0,C 180,E1 -31182.313,E2 -31182.313} C_VEL
LIN {X 0,Y 226.13,Z 975.682,A -85,B 0,C 180,E1 -31183.589,E2 -31183.589} C_VEL
LIN {X 0,Y 230.321,Z 985.854,A -85,B 0,C 180,E1 -31187.738,E2 -31187.738} C_VEL
LIN {X 0,Y 232.536,Z 988.183,A -85,B 0,C 180,E1 -31188.967,E2 -31188.967} C_VEL
LIN {X 0,Y 243.874,Z 996.291,A -85,B 0,C 180,E1 -31193.794,E2 -31193.794} C_VEL
LIN {X 0,Y 251.598,Z 1002.083,A -85,B 0,C 180,E1 -31196.929,E2 -31196.929} C_VEL
LIN {X 0,Y 257.412,Z 1006.318,A -85,B 0,C 180,E1 -31199.318,E2 -31199.318} C_VEL
LIN {X 0,Y 263.046,Z 1010.664,A -85,B 0,C 180,E1 -31201.845,E2 -31201.845} C_VEL
LIN {X 0,Y 266.839,Z 1013.308,A -85,B 0,C 180,E1 -31203.57,E2 -31203.57} C_VEL
LIN {X 0,Y 270.576,Z 1016.025,A -85,B 0,C 180,E1 -31205.444,E2 -31205.444} C_VEL
LIN {X 0,Y 275.19,Z 1019.344,A -85,B 0,C 180,E1 -31207.959,E2 -31207.959} C_VEL
LIN {X 0,Y 277.747,Z 1021.098,A -85,B 0,C 180,E1 -31209.426,E2 -31209.426} C_VEL
LIN {X 0,Y 282.706,Z 1024.578,A -85,B 0,C 180,E1 -31212.644,E2 -31212.644} C_VEL
LIN {X 0,Y 286.606,Z 1027.448,A -85,B 0,C 180,E1 -31215.806,E2 -31215.806} C_VEL
LIN {X 0,Y 289.892,Z 1029.539,A -85,B 0,C 180,E1 -31218.817,E2 -31218.817} C_VEL
LIN {X 0,Y 292.598,Z 1030.846,A -85,B 0,C 180,E1 -31221.714,E2 -31221.714} C_VEL
LIN {X 0,Y 294.589,Z 1031.745,A -85,B 0,C 180,E1 -31224.524,E2 -31224.524} C_VEL
LIN {X 0,Y 295.76,Z 1032.302,A -85,B 0,C 180,E1 -31227.276,E2 -31227.276} C_VEL
LIN {X 0,Y 296.099,Z 1032.451,A -85,B 0,C 180,E1 -31230,E2 -31230} C_VEL
LIN {X 0,Y 295.76,Z 1032.297,A -85,B 0,C 180,E1 -31232.724,E2 -31232.724} C_VEL
LIN {X 0,Y 294.523,Z 1031.786,A -85,B 0,C 180,E1 -31235.477,E2 -31235.477} C_VEL
LIN {X 0,Y 292.598,Z 1030.851,A -85,B 0,C 180,E1 -31238.286,E2 -31238.286} C_VEL
LIN {X 0,Y 289.892,Z 1029.537,A -85,B 0,C 180,E1 -31241.183,E2 -31241.183} C_VEL
LIN {X 0,Y 286.606,Z 1027.446,A -85,B 0,C 180,E1 -31244.194,E2 -31244.194} C_VEL
LIN {X 0,Y 282.745,Z 1024.558,A -85,B 0,C 180,E1 -31247.354,E2 -31247.354} C_VEL
LIN {X 0,Y 280.225,Z 1022.803,A -85,B 0,C 180,E1 -31249.028,E2 -31249.028} C_VEL
LIN {X 0,Y 277.444,Z 1020.855,A -85,B 0,C 180,E1 -31250.771,E2 -31250.771} C_VEL
LIN {X 0,Y 272.721,Z 1017.562,A -85,B 0,C 180,E1 -31253.421,E2 -31253.421} C_VEL
LIN {X 0,Y 269.456,Z 1015.109,A -85,B 0,C 180,E1 -31255.161,E2 -31255.161} C_VEL
LIN {X 0,Y 264.99,Z 1011.994,A -85,B 0,C 180,E1 -31257.296,E2 -31257.296} C_VEL
LIN {X 0,Y 259.292,Z 1007.843,A -85,B 0,C 180,E1 -31259.85,E2 -31259.85} C_VEL
LIN {X 0,Y 255.528,Z 1004.956,A -85,B 0,C 180,E1 -31261.504,E2 -31261.504} C_VEL
LIN {X 0,Y 245.669,Z 997.558,A -85,B 0,C 180,E1 -31265.491,E2 -31265.491} C_VEL
LIN {X 0,Y 236.326,Z 990.89,A -85,B 0,C 180,E1 -31269.359,E2 -31269.359} C_VEL
LIN {X 0,Y 223.973,Z 981.975,A -85,B 0,C 180,E1 -31275.089,E2 -31275.089} C_VEL
LIN {X 0,Y 209.517,Z 969.116,A -85,B 0,C 180,E1 -31283.937,E2 -31283.937} C_VEL
LIN {X 0,Y 202.167,Z 958.924,A -85,B 0,C 180,E1 -31290.878,E2 -31290.878} C_VEL
LIN {X 0,Y 197.881,Z 947.737,A -85,B 0,C 180,E1 -31297.995,E2 -31297.995} C_VEL
LIN {X 0,Y 196.562,Z 936.363,A -85,B 0,C 180,E1 -31304.447,E2 -31304.447} C_VEL
LIN {X 0,Y 197.127,Z 925.945,A -85,B 0,C 180,E1 -31309.732,E2 -31309.732} C_VEL
LIN {X 0,Y 197.599,Z 922.062,A -85,B 0,C 180,E1 -31311.564,E2 -31311.564} C_VEL
LIN {X 0,Y 195.489,Z 927.652,A -85,B 0,C 180,E1 -31311.635,E2 -31311.635} C_VEL
LIN {X 0,Y 188.237,Z 943.777,A -85,B 0,C 180,E1 -31311.641,E2 -31311.641} C_VEL
LIN {X 0,Y 180.216,Z 958.165,A -85,B 0,C 180,E1 -31311.704,E2 -31311.704} C_VEL
LIN {X 0,Y 172.21,Z 970.396,A -85,B 0,C 180,E1 -31311.743,E2 -31311.743} C_VEL
LIN {X 0,Y 164.195,Z 981.009,A -85,B 0,C 180,E1 -31311.803,E2 -31311.803} C_VEL
LIN {X 0,Y 155.198,Z 991.459,A -85,B 0,C 180,E1 -31311.888,E2 -31311.888} C_VEL
LIN {X 0,Y 147.249,Z 999.665,A -85,B 0,C 180,E1 -31312.031,E2 -31312.031} C_VEL
LIN {X 0,Y 136.553,Z 1009.385,A -85,B 0,C 180,E1 -31312.188,E2 -31312.188} C_VEL
LIN {X 0,Y 125.853,Z 1017.893,A -85,B 0,C 180,E1 -31312.388,E2 -31312.388} C_VEL
LIN {X 0,Y 113.359,Z 1026.486,A -85,B 0,C 180,E1 -31312.718,E2 -31312.718} C_VEL
LIN {X 0,Y 102.642,Z 1032.911,A -85,B 0,C 180,E1 -31313.121,E2 -31313.121} C_VEL
LIN {X 0,Y 88.373,Z 1040.173,A -85,B 0,C 180,E1 -31313.75,E2 -31313.75} C_VEL
LIN {X 0,Y 77.68,Z 1044.822,A -85,B 0,C 180,E1 -31314.377,E2 -31314.377} C_VEL
LIN {X 0,Y 63.437,Z 1049.935,A -85,B 0,C 180,E1 -31315.606,E2 -31315.606} C_VEL
LIN {X 0,Y 49.244,Z 1053.951,A -85,B 0,C 180,E1 -31317.442,E2 -31317.442} C_VEL
LIN {X 0,Y 35.141,Z 1056.932,A -85,B 0,C 180,E1 -31320.623,E2 -31320.623} C_VEL
LIN {X 0,Y 28.157,Z 1058.134,A -85,B 0,C 180,E1 -31323.262,E2 -31323.262} C_VEL
LIN {X 0,Y 14.576,Z 1059.638,A -85,B 0,C 180,E1 -31335.35,E2 -31335.35} C_VEL
LIN {X 0,Y 5.638,Z 1060.168,A -85,B 0,C 180,E1 -31410,E2 -31410} C_VEL
LIN {X 0,Y 14.576,Z 1059.638,A -85,B 0,C 180,E1 -31484.649,E2 -31484.649} C_VEL
LIN {X 0,Y 28.158,Z 1058.134,A -85,B 0,C 180,E1 -31496.705,E2 -31496.705} C_VEL
LIN {X 0,Y 42.176,Z 1055.637,A -85,B 0,C 180,E1 -31501.19,E2 -31501.19} C_VEL
LIN {X 0,Y 59.884,Z 1051.026,A -85,B 0,C 180,E1 -31504.023,E2 -31504.023} C_VEL
LIN {X 0,Y 70.554,Z 1047.524,A -85,B 0,C 180,E1 -31505.072,E2 -31505.072} C_VEL
LIN {X 0,Y 84.808,Z 1041.795,A -85,B 0,C 180,E1 -31506.06,E2 -31506.06} C_VEL
LIN {X 0,Y 95.504,Z 1036.733,A -85,B 0,C 180,E1 -31506.575,E2 -31506.575} C_VEL
LIN {X 0,Y 108.965,Z 1029.217,A -85,B 0,C 180,E1 -31507.117,E2 -31507.117} C_VEL
LIN {X 0,Y 120.499,Z 1021.728,A -85,B 0,C 180,E1 -31507.484,E2 -31507.484} C_VEL
LIN {X 0,Y 131.217,Z 1013.772,A -85,B 0,C 180,E1 -31507.764,E2 -31507.764} C_VEL
LIN {X 0,Y 141.896,Z 1004.674,A -85,B 0,C 180,E1 -31507.879,E2 -31507.879} C_VEL
LIN {X 0,Y 151.421,Z 995.492,A -85,B 0,C 180,E1 -31508.068,E2 -31508.068} C_VEL
LIN {X 0,Y 161.522,Z 984.268,A -85,B 0,C 180,E1 -31508.169,E2 -31508.169} C_VEL
LIN {X 0,Y 170.432,Z 972.885,A -85,B 0,C 180,E1 -31508.252,E2 -31508.252} C_VEL
LIN {X 0,Y 178.438,Z 961.037,A -85,B 0,C 180,E1 -31508.29,E2 -31508.29} C_VEL
LIN {X 0,Y 185.526,Z 948.876,A -85,B 0,C 180,E1 -31508.346,E2 -31508.346} C_VEL
LIN {X 0,Y 191.796,Z 936.188,A -85,B 0,C 180,E1 -31508.374,E2 -31508.374} C_VEL
LIN {X 0,Y 196.979,Z 923.653,A -85,B 0,C 180,E1 -31508.374,E2 -31508.374} C_VEL
LIN {X 0,Y 197.605,Z 922.046,A -85,B 0,C 180,E1 -31508.435,E2 -31508.435} C_VEL
LIN {X 0,Y 196.621,Z 932.34,A -85,B 0,C 180,E1 -31513.434,E2 -31513.434} C_VEL
LIN {X 0,Y 196.956,Z 942.17,A -85,B 0,C 180,E1 -31518.732,E2 -31518.732} C_VEL
LIN {X 0,Y 199.779,Z 953.705,A -85,B 0,C 180,E1 -31525.709,E2 -31525.709} C_VEL
LIN {X 0,Y 205.985,Z 964.792,A -85,B 0,C 180,E1 -31533.086,E2 -31533.086} C_VEL
LIN {X 0,Y 217.601,Z 976.88,A -85,B 0,C 180,E1 -31541.459,E2 -31541.459} C_VEL
LIN {X 0,Y 230.869,Z 987.035,A -85,B 0,C 180,E1 -31548.227,E2 -31548.227} C_VEL
LIN {X 0,Y 232.536,Z 988.183,A -85,B 0,C 180,E1 -31548.967,E2 -31548.967} C_VEL
LIN {X 0,Y 234.765,Z 990.511,A -85,B 0,C 180,E1 -31550.184,E2 -31550.184} C_VEL
LIN {X 0,Y 236.977,Z 995.457,A -85,B 0,C 180,E1 -31552.209,E2 -31552.209} C_VEL
LIN {X 0,Y 239.191,Z 1000.383,A -85,B 0,C 180,E1 -31554.232,E2 -31554.232} C_VEL
LIN {X 0,Y 241.424,Z 1002.686,A -85,B 0,C 180,E1 -31555.42,E2 -31555.42} C_VEL
LIN {X 0,Y 250.576,Z 1009.373,A -85,B 0,C 180,E1 -31559.201,E2 -31559.201} C_VEL
LIN {X 0,Y 255.82,Z 1013.377,A -85,B 0,C 180,E1 -31561.534,E2 -31561.534} C_VEL
LIN {X 0,Y 259.679,Z 1016.15,A -85,B 0,C 180,E1 -31563.266,E2 -31563.266} C_VEL
LIN {X 0,Y 263.449,Z 1018.833,A -85,B 0,C 180,E1 -31565.094,E2 -31565.094} C_VEL
LIN {X 0,Y 268.107,Z 1022.208,A -85,B 0,C 180,E1 -31567.587,E2 -31567.587} C_VEL
LIN {X 0,Y 270.81,Z 1024.096,A -85,B 0,C 180,E1 -31569.107,E2 -31569.107} C_VEL
LIN {X 0,Y 275.716,Z 1027.506,A -85,B 0,C 180,E1 -31572.189,E2 -31572.189} C_VEL
LIN {X 0,Y 277.974,Z 1029.17,A -85,B 0,C 180,E1 -31573.891,E2 -31573.891} C_VEL
LIN {X 0,Y 281.715,Z 1031.832,A -85,B 0,C 180,E1 -31577.025,E2 -31577.025} C_VEL
LIN {X 0,Y 285.151,Z 1033.762,A -85,B 0,C 180,E1 -31580.35,E2 -31580.35} C_VEL
LIN {X 0,Y 287.36,Z 1034.816,A -85,B 0,C 180,E1 -31582.976,E2 -31582.976} C_VEL
LIN {X 0,Y 288.973,Z 1035.574,A -85,B 0,C 180,E1 -31585.659,E2 -31585.659} C_VEL
LIN {X 0,Y 289.578,Z 1035.782,A -85,B 0,C 180,E1 -31587.218,E2 -31587.218} C_VEL
LIN {X 0,Y 289.93,Z 1035.941,A -85,B 0,C 180,E1 -31590,E2 -31590} C_VEL
LIN {X 0,Y 289.538,Z 1035.8,A -85,B 0,C 180,E1 -31592.783,E2 -31592.783} C_VEL
LIN {X 0,Y 288.274,Z 1035.286,A -85,B 0,C 180,E1 -31595.596,E2 -31595.596} C_VEL
LIN {X 0,Y 286.223,Z 1034.262,A -85,B 0,C 180,E1 -31598.472,E2 -31598.472} C_VEL
LIN {X 0,Y 283.337,Z 1032.815,A -85,B 0,C 180,E1 -31601.445,E2 -31601.445} C_VEL
LIN {X 0,Y 281.485,Z 1031.687,A -85,B 0,C 180,E1 -31603.164,E2 -31603.164} C_VEL
LIN {X 0,Y 277.924,Z 1029.126,A -85,B 0,C 180,E1 -31606.15,E2 -31606.15} C_VEL
LIN {X 0,Y 274.461,Z 1026.58,A -85,B 0,C 180,E1 -31608.661,E2 -31608.661} C_VEL
LIN {X 0,Y 269.987,Z 1023.529,A -85,B 0,C 180,E1 -31611.372,E2 -31611.372} C_VEL
LIN {X 0,Y 265.51,Z 1020.32,A -85,B 0,C 180,E1 -31613.84,E2 -31613.84} C_VEL
LIN {X 0,Y 261.436,Z 1017.313,A -85,B 0,C 180,E1 -31615.925,E2 -31615.925} C_VEL
LIN {X 0,Y 255.825,Z 1013.402,A -85,B 0,C 180,E1 -31618.468,E2 -31618.468} C_VEL
LIN {X 0,Y 250.615,Z 1009.404,A -85,B 0,C 180,E1 -31620.781,E2 -31620.781} C_VEL
LIN {X 0,Y 242.257,Z 1003.299,A -85,B 0,C 180,E1 -31624.23,E2 -31624.23} C_VEL
LIN {X 0,Y 232.761,Z 996.57,A -85,B 0,C 180,E1 -31628.276,E2 -31628.276} C_VEL
LIN {X 0,Y 220.297,Z 987.891,A -85,B 0,C 180,E1 -31634.128,E2 -31634.128} C_VEL
LIN {X 0,Y 205.857,Z 975.553,A -85,B 0,C 180,E1 -31643.102,E2 -31643.102} C_VEL
LIN {X 0,Y 197.632,Z 964.15,A -85,B 0,C 180,E1 -31651.311,E2 -31651.311} C_VEL
LIN {X 0,Y 193.867,Z 952.984,A -85,B 0,C 180,E1 -31658.746,E2 -31658.746} C_VEL
LIN {X 0,Y 193.202,Z 941.965,A -85,B 0,C 180,E1 -31665.249,E2 -31665.249} C_VEL
LIN {X 0,Y 193.904,Z 933.868,A -85,B 0,C 180,E1 -31669.56,E2 -31669.56} C_VEL
LIN {X 0,Y 188.548,Z 945.184,A -85,B 0,C 180,E1 -31669.508,E2 -31669.508} C_VEL
LIN {X 0,Y 181.385,Z 957.963,A -85,B 0,C 180,E1 -31669.47,E2 -31669.47} C_VEL
LIN {X 0,Y 173.38,Z 970.195,A -85,B 0,C 180,E1 -31669.406,E2 -31669.406} C_VEL
LIN {X 0,Y 164.475,Z 981.891,A -85,B 0,C 180,E1 -31669.345,E2 -31669.345} C_VEL
LIN {X 0,Y 156.37,Z 991.257,A -85,B 0,C 180,E1 -31669.289,E2 -31669.289} C_VEL
LIN {X 0,Y 148.389,Z 999.49,A -85,B 0,C 180,E1 -31669.272,E2 -31669.272} C_VEL
LIN {X 0,Y 137.704,Z 1009.183,A -85,B 0,C 180,E1 -31669.245,E2 -31669.245} C_VEL
LIN {X 0,Y 127.003,Z 1017.689,A -85,B 0,C 180,E1 -31669.177,E2 -31669.177} C_VEL
LIN {X 0,Y 114.489,Z 1026.282,A -85,B 0,C 180,E1 -31669.158,E2 -31669.158} C_VEL
LIN {X 0,Y 103.75,Z 1032.705,A -85,B 0,C 180,E1 -31669.172,E2 -31669.172} C_VEL
LIN {X 0,Y 89.444,Z 1039.968,A -85,B 0,C 180,E1 -31669.16,E2 -31669.16} C_VEL
LIN {X 0,Y 78.713,Z 1044.615,A -85,B 0,C 180,E1 -31669.148,E2 -31669.148} C_VEL
LIN {X 0,Y 64.394,Z 1049.729,A -85,B 0,C 180,E1 -31669.185,E2 -31669.185} C_VEL
LIN {X 0,Y 50.085,Z 1053.745,A -85,B 0,C 180,E1 -31669.179,E2 -31669.179} C_VEL
LIN {X 0,Y 35.795,Z 1056.725,A -85,B 0,C 180,E1 -31669.013,E2 -31669.013} C_VEL
LIN {X 0,Y 28.663,Z 1057.927,A -85,B 0,C 180,E1 -31668.743,E2 -31668.743} C_VEL
LIN {X 0,Y 14.443,Z 1059.429,A -85,B 0,C 180,E1 -31666.697,E2 -31666.697} C_VEL
LIN {X 0,Y 1.494,Z 1059.962,A -85,B 0,C 180,E1 -31590,E2 -31590} C_VEL
LIN {X 0,Y 14.443,Z 1059.429,A -85,B 0,C 180,E1 -31513.3,E2 -31513.3} C_VEL
LIN {X 0,Y 28.659,Z 1057.928,A -85,B 0,C 180,E1 -31511.221,E2 -31511.221} C_VEL
LIN {X 0,Y 42.936,Z 1055.431,A -85,B 0,C 180,E1 -31510.864,E2 -31510.864} C_VEL
LIN {X 0,Y 60.815,Z 1050.821,A -85,B 0,C 180,E1 -31510.806,E2 -31510.806} C_VEL
LIN {X 0,Y 71.558,Z 1047.317,A -85,B 0,C 180,E1 -31510.851,E2 -31510.851} C_VEL
LIN {X 0,Y 85.865,Z 1041.59,A -85,B 0,C 180,E1 -31510.838,E2 -31510.838} C_VEL
LIN {X 0,Y 96.589,Z 1036.528,A -85,B 0,C 180,E1 -31510.81,E2 -31510.81} C_VEL
LIN {X 0,Y 110.616,Z 1028.687,A -85,B 0,C 180,E1 -31510.848,E2 -31510.848} C_VEL
LIN {X 0,Y 121.644,Z 1021.523,A -85,B 0,C 180,E1 -31510.841,E2 -31510.841} C_VEL
LIN {X 0,Y 132.378,Z 1013.568,A -85,B 0,C 180,E1 -31510.844,E2 -31510.844} C_VEL
LIN {X 0,Y 143.05,Z 1004.471,A -85,B 0,C 180,E1 -31510.714,E2 -31510.714} C_VEL
LIN {X 0,Y 152.798,Z 995.066,A -85,B 0,C 180,E1 -31510.726,E2 -31510.726} C_VEL
LIN {X 0,Y 162.691,Z 984.064,A -85,B 0,C 180,E1 -31510.662,E2 -31510.662} C_VEL
LIN {X 0,Y 171.601,Z 972.684,A -85,B 0,C 180,E1 -31510.609,E2 -31510.609} C_VEL
LIN {X 0,Y 179.601,Z 960.836,A -85,B 0,C 180,E1 -31510.534,E2 -31510.534} C_VEL
LIN {X 0,Y 186.624,Z 948.807,A -85,B 0,C 180,E1 -31510.509,E2 -31510.509} C_VEL
LIN {X 0,Y 192.962,Z 935.989,A -85,B 0,C 180,E1 -31510.468,E2 -31510.468} C_VEL
LIN {X 0,Y 193.823,Z 934.051,A -85,B 0,C 180,E1 -31510.445,E2 -31510.445} C_VEL
LIN {X 0,Y 193.108,Z 945.812,A -85,B 0,C 180,E1 -31516.926,E2 -31516.926} C_VEL
LIN {X 0,Y 194.55,Z 956.386,A -85,B 0,C 180,E1 -31523.413,E2 -31523.413} C_VEL
LIN {X 0,Y 199.196,Z 966.929,A -85,B 0,C 180,E1 -31530.662,E2 -31530.662} C_VEL
LIN {X 0,Y 208.266,Z 978.084,A -85,B 0,C 180,E1 -31538.753,E2 -31538.753} C_VEL
LIN {X 0,Y 221.987,Z 989.117,A -85,B 0,C 180,E1 -31546.732,E2 -31546.732} C_VEL
LIN {X 0,Y 230.905,Z 995.316,A -85,B 0,C 180,E1 -31550.907,E2 -31550.907} C_VEL
LIN {X 0,Y 240.34,Z 1001.899,A -85,B 0,C 180,E1 -31554.961,E2 -31554.961} C_VEL
LIN {X 0,Y 241.424,Z 1002.686,A -85,B 0,C 180,E1 -31555.42,E2 -31555.42} C_VEL
LIN {X 0,Y 243.612,Z 1005.089,A -85,B 0,C 180,E1 -31556.593,E2 -31556.593} C_VEL
LIN {X 0,Y 245.638,Z 1009.821,A -85,B 0,C 180,E1 -31558.582,E2 -31558.582} C_VEL
LIN {X 0,Y 247.08,Z 1013.581,A -85,B 0,C 180,E1 -31560.19,E2 -31560.19} C_VEL
LIN {X 0,Y 248.806,Z 1016.018,A -85,B 0,C 180,E1 -31561.384,E2 -31561.384} C_VEL
LIN {X 0,Y 249.596,Z 1016.688,A -85,B 0,C 180,E1 -31561.773,E2 -31561.773} C_VEL
LIN {X 0,Y 253.859,Z 1019.717,A -85,B 0,C 180,E1 -31563.708,E2 -31563.708} C_VEL
LIN {X 0,Y 258.39,Z 1022.995,A -85,B 0,C 180,E1 -31565.922,E2 -31565.922} C_VEL
LIN {X 0,Y 263.759,Z 1026.811,A -85,B 0,C 180,E1 -31568.841,E2 -31568.841} C_VEL
LIN {X 0,Y 268.423,Z 1030.057,A -85,B 0,C 180,E1 -31571.689,E2 -31571.689} C_VEL
LIN {X 0,Y 271.074,Z 1031.962,A -85,B 0,C 180,E1 -31573.59,E2 -31573.59} C_VEL
LIN {X 0,Y 274.871,Z 1034.695,A -85,B 0,C 180,E1 -31576.697,E2 -31576.697} C_VEL
LIN {X 0,Y 278.344,Z 1036.723,A -85,B 0,C 180,E1 -31579.967,E2 -31579.967} C_VEL
LIN {X 0,Y 280.853,Z 1037.979,A -85,B 0,C 180,E1 -31582.813,E2 -31582.813} C_VEL
LIN {X 0,Y 282.226,Z 1038.558,A -85,B 0,C 180,E1 -31584.917,E2 -31584.917} C_VEL
LIN {X 0,Y 283.215,Z 1038.965,A -85,B 0,C 180,E1 -31587.155,E2 -31587.155} C_VEL
LIN {X 0,Y 283.604,Z 1039.139,A -85,B 0,C 180,E1 -31590,E2 -31590} C_VEL
LIN {X 0,Y 283.161,Z 1038.988,A -85,B 0,C 180,E1 -31592.845,E2 -31592.845} C_VEL
LIN {X 0,Y 282.2,Z 1038.602,A -85,B 0,C 180,E1 -31595.025,E2 -31595.025} C_VEL
LIN {X 0,Y 280.849,Z 1037.984,A -85,B 0,C 180,E1 -31597.188,E2 -31597.188} C_VEL
LIN {X 0,Y 278.344,Z 1036.729,A -85,B 0,C 180,E1 -31600.033,E2 -31600.033} C_VEL
LIN {X 0,Y 274.871,Z 1034.693,A -85,B 0,C 180,E1 -31603.303,E2 -31603.303} C_VEL
LIN {X 0,Y 271.085,Z 1031.949,A -85,B 0,C 180,E1 -31606.418,E2 -31606.418} C_VEL
LIN {X 0,Y 267.477,Z 1029.37,A -85,B 0,C 180,E1 -31608.934,E2 -31608.934} C_VEL
LIN {X 0,Y 262.207,Z 1025.721,A -85,B 0,C 180,E1 -31612.039,E2 -31612.039} C_VEL
LIN {X 0,Y 256.276,Z 1021.36,A -85,B 0,C 180,E1 -31615.182,E2 -31615.182} C_VEL
LIN {X 0,Y 250.415,Z 1017.296,A -85,B 0,C 180,E1 -31617.866,E2 -31617.866} C_VEL
LIN {X 0,Y 244.583,Z 1012.872,A -85,B 0,C 180,E1 -31620.455,E2 -31620.455} C_VEL
LIN {X 0,Y 234.679,Z 1005.889,A -85,B 0,C 180,E1 -31624.679,E2 -31624.679} C_VEL
LIN {X 0,Y 225.406,Z 999.615,A -85,B 0,C 180,E1 -31628.788,E2 -31628.788} C_VEL
LIN {X 0,Y 213.826,Z 991.685,A -85,B 0,C 180,E1 -31634.53,E2 -31634.53} C_VEL
LIN {X 0,Y 200.47,Z 980.169,A -85,B 0,C 180,E1 -31643.418,E2 -31643.418} C_VEL
LIN {X 0,Y 193.715,Z 970.893,A -85,B 0,C 180,E1 -31650.54,E2 -31650.54} C_VEL
LIN {X 0,Y 189.961,Z 959.926,A -85,B 0,C 180,E1 -31658.287,E2 -31658.287} C_VEL
LIN {X 0,Y 189.458,Z 949.396,A -85,B 0,C 180,E1 -31664.95,E2 -31664.95} C_VEL
LIN {X 0,Y 189.841,Z 945.529,A -85,B 0,C 180,E1 -31667.167,E2 -31667.167} C_VEL
LIN {X 0,Y 189.144,Z 946.551,A -85,B 0,C 180,E1 -31667.377,E2 -31667.377} C_VEL
LIN {X 0,Y 181.931,Z 959.198,A -85,B 0,C 180,E1 -31667.26,E2 -31667.26} C_VEL
LIN {X 0,Y 174.828,Z 969.994,A -85,B 0,C 180,E1 -31667.113,E2 -31667.113} C_VEL
LIN {X 0,Y 165.948,Z 981.688,A -85,B 0,C 180,E1 -31666.916,E2 -31666.916} C_VEL
LIN {X 0,Y 157.057,Z 991.911,A -85,B 0,C 180,E1 -31666.716,E2 -31666.716} C_VEL
LIN {X 0,Y 147.67,Z 1001.349,A -85,B 0,C 180,E1 -31666.56,E2 -31666.56} C_VEL
LIN {X 0,Y 137.445,Z 1010.442,A -85,B 0,C 180,E1 -31666.288,E2 -31666.288} C_VEL
LIN {X 0,Y 126.764,Z 1018.762,A -85,B 0,C 180,E1 -31665.977,E2 -31665.977} C_VEL
LIN {X 0,Y 116.057,Z 1026.078,A -85,B 0,C 180,E1 -31665.667,E2 -31665.667} C_VEL
LIN {X 0,Y 105.342,Z 1032.499,A -85,B 0,C 180,E1 -31665.321,E2 -31665.321} C_VEL
LIN {X 0,Y 91.076,Z 1039.762,A -85,B 0,C 180,E1 -31664.699,E2 -31664.699} C_VEL
LIN {X 0,Y 80.379,Z 1044.409,A -85,B 0,C 180,E1 -31664.106,E2 -31664.106} C_VEL
LIN {X 0,Y 66.133,Z 1049.523,A -85,B 0,C 180,E1 -31663.021,E2 -31663.021} C_VEL
LIN {X 0,Y 51.93,Z 1053.538,A -85,B 0,C 180,E1 -31661.319,E2 -31661.319} C_VEL
LIN {X 0,Y 37.831,Z 1056.52,A -85,B 0,C 180,E1 -31658.257,E2 -31658.257} C_VEL
LIN {X 0,Y 30.883,Z 1057.72,A -85,B 0,C 180,E1 -31655.541,E2 -31655.541} C_VEL
LIN {X 0,Y 17.549,Z 1059.219,A -85,B 0,C 180,E1 -31643.22,E2 -31643.22} C_VEL
LIN {X 0,Y 8.637,Z 1059.755,A -85,B 0,C 180,E1 -31590,E2 -31590} C_VEL
LIN {X 0,Y 17.548,Z 1059.219,A -85,B 0,C 180,E1 -31536.776,E2 -31536.776} C_VEL
LIN {X 0,Y 30.874,Z 1057.721,A -85,B 0,C 180,E1 -31524.424,E2 -31524.424} C_VEL
LIN {X 0,Y 44.855,Z 1055.222,A -85,B 0,C 180,E1 -31519.938,E2 -31519.938} C_VEL
LIN {X 0,Y 62.57,Z 1050.615,A -85,B 0,C 180,E1 -31517.31,E2 -31517.31} C_VEL
LIN {X 0,Y 75.2,Z 1046.376,A -85,B 0,C 180,E1 -31516.281,E2 -31516.281} C_VEL
LIN {X 0,Y 87.508,Z 1041.385,A -85,B 0,C 180,E1 -31515.48,E2 -31515.48} C_VEL
LIN {X 0,Y 98.2,Z 1036.321,A -85,B 0,C 180,E1 -31514.95,E2 -31514.95} C_VEL
LIN {X 0,Y 112.59,Z 1028.239,A -85,B 0,C 180,E1 -31514.458,E2 -31514.458} C_VEL
LIN {X 0,Y 124.982,Z 1020.04,A -85,B 0,C 180,E1 -31514.075,E2 -31514.075} C_VEL
LIN {X 0,Y 135.693,Z 1011.901,A -85,B 0,C 180,E1 -31513.808,E2 -31513.808} C_VEL
LIN {X 0,Y 146.023,Z 1002.896,A -85,B 0,C 180,E1 -31513.483,E2 -31513.483} C_VEL
LIN {X 0,Y 153.492,Z 995.717,A -85,B 0,C 180,E1 -31513.356,E2 -31513.356} C_VEL
LIN {X 0,Y 164.169,Z 983.86,A -85,B 0,C 180,E1 -31513.122,E2 -31513.122} C_VEL
LIN {X 0,Y 173.053,Z 972.484,A -85,B 0,C 180,E1 -31512.927,E2 -31512.927} C_VEL
LIN {X 0,Y 181.044,Z 960.634,A -85,B 0,C 180,E1 -31512.758,E2 -31512.758} C_VEL
LIN {X 0,Y 188.473,Z 947.811,A -85,B 0,C 180,E1 -31512.631,E2 -31512.631} C_VEL
LIN {X 0,Y 189.145,Z 946.553,A -85,B 0,C 180,E1 -31512.624,E2 -31512.624} C_VEL
LIN {X 0,Y 189.843,Z 945.525,A -85,B 0,C 180,E1 -31512.833,E2 -31512.833} C_VEL
LIN {X 0,Y 189.457,Z 954.328,A -85,B 0,C 180,E1 -31518.073,E2 -31518.073} C_VEL
LIN {X 0,Y 190.675,Z 963.255,A -85,B 0,C 180,E1 -31523.918,E2 -31523.918} C_VEL
LIN {X 0,Y 196.232,Z 974.904,A -85,B 0,C 180,E1 -31532.494,E2 -31532.494} C_VEL
LIN {X 0,Y 207.836,Z 987.088,A -85,B 0,C 180,E1 -31541.934,E2 -31541.934} C_VEL
LIN {X 0,Y 221.761,Z 997.176,A -85,B 0,C 180,E1 -31549.516,E2 -31549.516} C_VEL
LIN {X 0,Y 232.904,Z 1004.68,A -85,B 0,C 180,E1 -31554.56,E2 -31554.56} C_VEL
LIN {X 0,Y 242.039,Z 1011.143,A -85,B 0,C 180,E1 -31558.49,E2 -31558.49} C_VEL
LIN {X 0,Y 248.473,Z 1015.83,A -85,B 0,C 180,E1 -31561.26,E2 -31561.26} C_VEL
LIN {X 0,Y 249.596,Z 1016.688,A -85,B 0,C 180,E1 -31561.773,E2 -31561.773} C_VEL
LIN {X 0,Y 251.513,Z 1018.898,A -85,B 0,C 180,E1 -31562.95,E2 -31562.95} C_VEL
LIN {X 0,Y 252.937,Z 1023,A -85,B 0,C 180,E1 -31564.975,E2 -31564.975} C_VEL
LIN {X 0,Y 253.85,Z 1026.197,A -85,B 0,C 180,E1 -31566.629,E2 -31566.629} C_VEL
LIN {X 0,Y 255.207,Z 1028.266,A -85,B 0,C 180,E1 -31567.86,E2 -31567.86} C_VEL
LIN {X 0,Y 255.887,Z 1028.757,A -85,B 0,C 180,E1 -31568.261,E2 -31568.261} C_VEL
LIN {X 0,Y 260.359,Z 1031.907,A -85,B 0,C 180,E1 -31570.867,E2 -31570.867} C_VEL
LIN {X 0,Y 264.077,Z 1034.479,A -85,B 0,C 180,E1 -31573.35,E2 -31573.35} C_VEL
LIN {X 0,Y 267.795,Z 1037.199,A -85,B 0,C 180,E1 -31576.338,E2 -31576.338} C_VEL
LIN {X 0,Y 271.449,Z 1039.422,A -85,B 0,C 180,E1 -31579.682,E2 -31579.682} C_VEL
LIN {X 0,Y 272.852,Z 1040.165,A -85,B 0,C 180,E1 -31581.11,E2 -31581.11} C_VEL
LIN {X 0,Y 275.248,Z 1041.25,A -85,B 0,C 180,E1 -31584.138,E2 -31584.138} C_VEL
LIN {X 0,Y 276.089,Z 1041.625,A -85,B 0,C 180,E1 -31585.62,E2 -31585.62} C_VEL
LIN {X 0,Y 276.687,Z 1041.858,A -85,B 0,C 180,E1 -31587.088,E2 -31587.088} C_VEL
LIN {X 0,Y 277.151,Z 1042.036,A -85,B 0,C 180,E1 -31590,E2 -31590} C_VEL
LIN {X 0,Y 276.643,Z 1041.874,A -85,B 0,C 180,E1 -31592.912,E2 -31592.912} C_VEL
LIN {X 0,Y 275.381,Z 1041.344,A -85,B 0,C 180,E1 -31595.555,E2 -31595.555} C_VEL
LIN {X 0,Y 274.141,Z 1040.792,A -85,B 0,C 180,E1 -31597.364,E2 -31597.364} C_VEL
LIN {X 0,Y 272.852,Z 1040.167,A -85,B 0,C 180,E1 -31598.89,E2 -31598.89} C_VEL
LIN {X 0,Y 269.635,Z 1038.368,A -85,B 0,C 180,E1 -31602.035,E2 -31602.035} C_VEL
LIN {X 0,Y 267.708,Z 1037.122,A -85,B 0,C 180,E1 -31603.753,E2 -31603.753} C_VEL
LIN {X 0,Y 264.084,Z 1034.476,A -85,B 0,C 180,E1 -31606.656,E2 -31606.656} C_VEL
LIN {X 0,Y 260.388,Z 1031.873,A -85,B 0,C 180,E1 -31609.152,E2 -31609.152} C_VEL
LIN {X 0,Y 256.597,Z 1029.239,A -85,B 0,C 180,E1 -31611.374,E2 -31611.374} C_VEL
LIN {X 0,Y 250.875,Z 1025.061,A -85,B 0,C 180,E1 -31614.436,E2 -31614.436} C_VEL
LIN {X 0,Y 246.918,Z 1022.287,A -85,B 0,C 180,E1 -31616.29,E2 -31616.29} C_VEL
LIN {X 0,Y 238.602,Z 1016.289,A -85,B 0,C 180,E1 -31620.048,E2 -31620.048} C_VEL
LIN {X 0,Y 229.24,Z 1009.931,A -85,B 0,C 180,E1 -31624.132,E2 -31624.132} C_VEL
LIN {X 0,Y 219.825,Z 1003.78,A -85,B 0,C 180,E1 -31628.439,E2 -31628.439} C_VEL
LIN {X 0,Y 207.697,Z 995.714,A -85,B 0,C 180,E1 -31634.718,E2 -31634.718} C_VEL
LIN {X 0,Y 194.139,Z 983.716,A -85,B 0,C 180,E1 -31644.606,E2 -31644.606} C_VEL
LIN {X 0,Y 187.568,Z 972.79,A -85,B 0,C 180,E1 -31653.281,E2 -31653.281} C_VEL
LIN {X 0,Y 185.412,Z 962.552,A -85,B 0,C 180,E1 -31660.728,E2 -31660.728} C_VEL
LIN {X 0,Y 185.57,Z 956.116,A -85,B 0,C 180,E1 -31664.947,E2 -31664.947} C_VEL
LIN {X 0,Y 184.625,Z 957.388,A -85,B 0,C 180,E1 -31665.122,E2 -31665.122} C_VEL
LIN {X 0,Y 176.552,Z 969.794,A -85,B 0,C 180,E1 -31664.861,E2 -31664.861} C_VEL
LIN {X 0,Y 167.711,Z 981.484,A -85,B 0,C 180,E1 -31664.536,E2 -31664.536} C_VEL
LIN {X 0,Y 158.852,Z 991.709,A -85,B 0,C 180,E1 -31664.206,E2 -31664.206} C_VEL
LIN {X 0,Y 149.164,Z 1001.467,A -85,B 0,C 180,E1 -31663.863,E2 -31663.863} C_VEL
LIN {X 0,Y 139.307,Z 1010.239,A -85,B 0,C 180,E1 -31663.439,E2 -31663.439} C_VEL
LIN {X 0,Y 128.69,Z 1018.557,A -85,B 0,C 180,E1 -31662.878,E2 -31662.878} C_VEL
LIN {X 0,Y 118.047,Z 1025.873,A -85,B 0,C 180,E1 -31662.278,E2 -31662.278} C_VEL
LIN {X 0,Y 107.396,Z 1032.293,A -85,B 0,C 180,E1 -31661.596,E2 -31661.596} C_VEL
LIN {X 0,Y 93.234,Z 1039.558,A -85,B 0,C 180,E1 -31660.43,E2 -31660.43} C_VEL
LIN {X 0,Y 82.646,Z 1044.202,A -85,B 0,C 180,E1 -31659.29,E2 -31659.29} C_VEL
LIN {X 0,Y 68.591,Z 1049.317,A -85,B 0,C 180,E1 -31657.241,E2 -31657.241} C_VEL
LIN {X 0,Y 54.67,Z 1053.332,A -85,B 0,C 180,E1 -31654.138,E2 -31654.138} C_VEL
LIN {X 0,Y 41.055,Z 1056.313,A -85,B 0,C 180,E1 -31648.86,E2 -31648.86} C_VEL
LIN {X 0,Y 34.483,Z 1057.514,A -85,B 0,C 180,E1 -31644.608,E2 -31644.608} C_VEL
LIN {X 0,Y 22.596,Z 1059.01,A -85,B 0,C 180,E1 -31628.466,E2 -31628.466} C_VEL
LIN {X 0,Y 15.766,Z 1059.549,A -85,B 0,C 180,E1 -31590,E2 -31590} C_VEL
LIN {X 0,Y 22.594,Z 1059.01,A -85,B 0,C 180,E1 -31551.53,E2 -31551.53} C_VEL
LIN {X 0,Y 34.469,Z 1057.514,A -85,B 0,C 180,E1 -31535.359,E2 -31535.359} C_VEL
LIN {X 0,Y 47.792,Z 1055.014,A -85,B 0,C 180,E1 -31528.08,E2 -31528.08} C_VEL
LIN {X 0,Y 65.088,Z 1050.409,A -85,B 0,C 180,E1 -31523.396,E2 -31523.396} C_VEL
LIN {X 0,Y 76.647,Z 1046.507,A -85,B 0,C 180,E1 -31521.515,E2 -31521.515} C_VEL
LIN {X 0,Y 89.697,Z 1041.18,A -85,B 0,C 180,E1 -31519.913,E2 -31519.913} C_VEL
LIN {X 0,Y 100.3,Z 1036.115,A -85,B 0,C 180,E1 -31518.929,E2 -31518.929} C_VEL
LIN {X 0,Y 113.692,Z 1028.601,A -85,B 0,C 180,E1 -31518.003,E2 -31518.003} C_VEL
LIN {X 0,Y 125.147,Z 1021.114,A -85,B 0,C 180,E1 -31517.319,E2 -31517.319} C_VEL
LIN {X 0,Y 135.808,Z 1013.161,A -85,B 0,C 180,E1 -31516.796,E2 -31516.796} C_VEL
LIN {X 0,Y 146.393,Z 1004.063,A -85,B 0,C 180,E1 -31516.234,E2 -31516.234} C_VEL
LIN {X 0,Y 155.304,Z 995.513,A -85,B 0,C 180,E1 -31515.929,E2 -31515.929} C_VEL
LIN {X 0,Y 165.939,Z 983.656,A -85,B 0,C 180,E1 -31515.527,E2 -31515.527} C_VEL
LIN {X 0,Y 174.787,Z 972.283,A -85,B 0,C 180,E1 -31515.206,E2 -31515.206} C_VEL
LIN {X 0,Y 182.75,Z 960.436,A -85,B 0,C 180,E1 -31514.942,E2 -31514.942} C_VEL
LIN {X 0,Y 184.641,Z 957.378,A -85,B 0,C 180,E1 -31514.89,E2 -31514.89} C_VEL
LIN {X 0,Y 185.566,Z 956.142,A -85,B 0,C 180,E1 -31515.068,E2 -31515.068} C_VEL
LIN {X 0,Y 186.034,Z 967.886,A -85,B 0,C 180,E1 -31523,E2 -31523} C_VEL
LIN {X 0,Y 190.306,Z 978.402,A -85,B 0,C 180,E1 -31531.132,E2 -31531.132} C_VEL
LIN {X 0,Y 198.892,Z 988.682,A -85,B 0,C 180,E1 -31539.496,E2 -31539.496} C_VEL
LIN {X 0,Y 210.982,Z 997.98,A -85,B 0,C 180,E1 -31547.124,E2 -31547.124} C_VEL
LIN {X 0,Y 221.651,Z 1005.02,A -85,B 0,C 180,E1 -31552.436,E2 -31552.436} C_VEL
LIN {X 0,Y 229.241,Z 1009.929,A -85,B 0,C 180,E1 -31555.868,E2 -31555.868} C_VEL
LIN {X 0,Y 238.608,Z 1016.289,A -85,B 0,C 180,E1 -31559.953,E2 -31559.953} C_VEL
LIN {X 0,Y 246.921,Z 1022.315,A -85,B 0,C 180,E1 -31563.709,E2 -31563.709} C_VEL
LIN {X 0,Y 250.828,Z 1025.112,A -85,B 0,C 180,E1 -31565.588,E2 -31565.588} C_VEL
LIN {X 0,Y 255.887,Z 1028.757,A -85,B 0,C 180,E1 -31568.261,E2 -31568.261} C_VEL
LIN {X 0,Y 257.43,Z 1030.527,A -85,B 0,C 180,E1 -31569.468,E2 -31569.468} C_VEL
LIN {X 0,Y 257.977,Z 1032.527,A -85,B 0,C 180,E1 -31570.706,E2 -31570.706} C_VEL
LIN {X 0,Y 258.149,Z 1036.448,A -85,B 0,C 180,E1 -31573.236,E2 -31573.236} C_VEL
LIN {X 0,Y 258.827,Z 1038.051,A -85,B 0,C 180,E1 -31574.516,E2 -31574.516} C_VEL
LIN {X 0,Y 259.271,Z 1038.411,A -85,B 0,C 180,E1 -31574.939,E2 -31574.939} C_VEL
LIN {X 0,Y 262.464,Z 1040.612,A -85,B 0,C 180,E1 -31577.631,E2 -31577.631} C_VEL
LIN {X 0,Y 264.492,Z 1041.817,A -85,B 0,C 180,E1 -31579.463,E2 -31579.463} C_VEL
LIN {X 0,Y 265.895,Z 1042.596,A -85,B 0,C 180,E1 -31580.875,E2 -31580.875} C_VEL
LIN {X 0,Y 268.478,Z 1043.771,A -85,B 0,C 180,E1 -31583.99,E2 -31583.99} C_VEL
LIN {X 0,Y 269.398,Z 1044.176,A -85,B 0,C 180,E1 -31585.511,E2 -31585.511} C_VEL
LIN {X 0,Y 270.047,Z 1044.437,A -85,B 0,C 180,E1 -31587.016,E2 -31587.016} C_VEL
LIN {X 0,Y 270.566,Z 1044.637,A -85,B 0,C 180,E1 -31590,E2 -31590} C_VEL
LIN {X 0,Y 269.992,Z 1044.454,A -85,B 0,C 180,E1 -31592.984,E2 -31592.984} C_VEL
LIN {X 0,Y 269.337,Z 1044.196,A -85,B 0,C 180,E1 -31594.49,E2 -31594.49} C_VEL
LIN {X 0,Y 268.425,Z 1043.794,A -85,B 0,C 180,E1 -31596.011,E2 -31596.011} C_VEL
LIN {X 0,Y 267.293,Z 1043.254,A -85,B 0,C 180,E1 -31597.554,E2 -31597.554} C_VEL
LIN {X 0,Y 264.492,Z 1041.819,A -85,B 0,C 180,E1 -31600.537,E2 -31600.537} C_VEL
LIN {X 0,Y 260.578,Z 1039.323,A -85,B 0,C 180,E1 -31604.048,E2 -31604.048} C_VEL
LIN {X 0,Y 256.994,Z 1036.715,A -85,B 0,C 180,E1 -31606.838,E2 -31606.838} C_VEL
LIN {X 0,Y 252.918,Z 1033.893,A -85,B 0,C 180,E1 -31609.478,E2 -31609.478} C_VEL
LIN {X 0,Y 247.399,Z 1029.995,A -85,B 0,C 180,E1 -31612.597,E2 -31612.597} C_VEL
LIN {X 0,Y 241.453,Z 1025.75,A -85,B 0,C 180,E1 -31615.537,E2 -31615.537} C_VEL
LIN {X 0,Y 233.437,Z 1020.162,A -85,B 0,C 180,E1 -31619.182,E2 -31619.182} C_VEL
LIN {X 0,Y 225.542,Z 1014.987,A -85,B 0,C 180,E1 -31622.72,E2 -31622.72} C_VEL
LIN {X 0,Y 217.916,Z 1010.111,A -85,B 0,C 180,E1 -31626.268,E2 -31626.268} C_VEL
LIN {X 0,Y 205.395,Z 1002.234,A -85,B 0,C 180,E1 -31632.638,E2 -31632.638} C_VEL
LIN {X 0,Y 191.01,Z 990.808,A -85,B 0,C 180,E1 -31642.621,E2 -31642.621} C_VEL
LIN {X 0,Y 183.63,Z 980.276,A -85,B 0,C 180,E1 -31651.672,E2 -31651.672} C_VEL
LIN {X 0,Y 181.165,Z 970.243,A -85,B 0,C 180,E1 -31659.566,E2 -31659.566} C_VEL
LIN {X 0,Y 181.169,Z 966.182,A -85,B 0,C 180,E1 -31662.505,E2 -31662.505} C_VEL
LIN {X 0,Y 179.798,Z 967.827,A -85,B 0,C 180,E1 -31662.708,E2 -31662.708} C_VEL
LIN {X 0,Y 170.632,Z 980.195,A -85,B 0,C 180,E1 -31662.26,E2 -31662.26} C_VEL
LIN {X 0,Y 160.951,Z 991.506,A -85,B 0,C 180,E1 -31661.75,E2 -31661.75} C_VEL
LIN {X 0,Y 150.949,Z 1001.609,A -85,B 0,C 180,E1 -31661.232,E2 -31661.232} C_VEL
LIN {X 0,Y 141.51,Z 1010.037,A -85,B 0,C 180,E1 -31660.665,E2 -31660.665} C_VEL
LIN {X 0,Y 130.988,Z 1018.353,A -85,B 0,C 180,E1 -31659.871,E2 -31659.871} C_VEL
LIN {X 0,Y 118.803,Z 1026.698,A -85,B 0,C 180,E1 -31658.871,E2 -31658.871} C_VEL
LIN {X 0,Y 106.369,Z 1033.998,A -85,B 0,C 180,E1 -31657.666,E2 -31657.666} C_VEL
LIN {X 0,Y 95.891,Z 1039.352,A -85,B 0,C 180,E1 -31656.365,E2 -31656.365} C_VEL
LIN {X 0,Y 85.467,Z 1043.995,A -85,B 0,C 180,E1 -31654.758,E2 -31654.758} C_VEL
LIN {X 0,Y 71.689,Z 1049.111,A -85,B 0,C 180,E1 -31651.92,E2 -31651.92} C_VEL
LIN {X 0,Y 58.171,Z 1053.127,A -85,B 0,C 180,E1 -31647.747,E2 -31647.747} C_VEL
LIN {X 0,Y 45.2,Z 1056.107,A -85,B 0,C 180,E1 -31641.024,E2 -31641.024} C_VEL
LIN {X 0,Y 39.083,Z 1057.307,A -85,B 0,C 180,E1 -31635.994,E2 -31635.994} C_VEL
LIN {X 0,Y 28.572,Z 1058.8,A -85,B 0,C 180,E1 -31619.468,E2 -31619.468} C_VEL
LIN {X 0,Y 22.888,Z 1059.343,A -85,B 0,C 180,E1 -31590,E2 -31590} C_VEL
LIN {X 0,Y 28.569,Z 1058.801,A -85,B 0,C 180,E1 -31560.528,E2 -31560.528} C_VEL
LIN {X 0,Y 39.067,Z 1057.307,A -85,B 0,C 180,E1 -31543.982,E2 -31543.982} C_VEL
LIN {X 0,Y 51.59,Z 1054.804,A -85,B 0,C 180,E1 -31535.18,E2 -31535.18} C_VEL
LIN {X 0,Y 68.276,Z 1050.204,A -85,B 0,C 180,E1 -31528.964,E2 -31528.964} C_VEL
LIN {X 0,Y 78.716,Z 1046.635,A -85,B 0,C 180,E1 -31526.512,E2 -31526.512} C_VEL
LIN {X 0,Y 92.404,Z 1040.975,A -85,B 0,C 180,E1 -31524.124,E2 -31524.124} C_VEL
LIN {X 0,Y 102.857,Z 1035.91,A -85,B 0,C 180,E1 -31522.721,E2 -31522.721} C_VEL
LIN {X 0,Y 115.243,Z 1028.949,A -85,B 0,C 180,E1 -31521.462,E2 -31521.462} C_VEL
LIN {X 0,Y 127.471,Z 1020.909,A -85,B 0,C 180,E1 -31520.405,E2 -31520.405} C_VEL
LIN {X 0,Y 138.05,Z 1012.957,A -85,B 0,C 180,E1 -31519.645,E2 -31519.645} C_VEL
LIN {X 0,Y 148.561,Z 1003.859,A -85,B 0,C 180,E1 -31518.894,E2 -31518.894} C_VEL
LIN {X 0,Y 157.422,Z 995.306,A -85,B 0,C 180,E1 -31518.438,E2 -31518.438} C_VEL
LIN {X 0,Y 167.992,Z 983.452,A -85,B 0,C 180,E1 -31517.876,E2 -31517.876} C_VEL
LIN {X 0,Y 176.794,Z 972.082,A -85,B 0,C 180,E1 -31517.44,E2 -31517.44} C_VEL
LIN {X 0,Y 179.798,Z 967.826,A -85,B 0,C 180,E1 -31517.292,E2 -31517.292} C_VEL
LIN {X 0,Y 181.189,Z 966.151,A -85,B 0,C 180,E1 -31517.493,E2 -31517.493} C_VEL
LIN {X 0,Y 181.881,Z 974.849,A -85,B 0,C 180,E1 -31523.936,E2 -31523.936} C_VEL
LIN {X 0,Y 186.95,Z 985.947,A -85,B 0,C 180,E1 -31533.126,E2 -31533.126} C_VEL
LIN {X 0,Y 197.562,Z 996.63,A -85,B 0,C 180,E1 -31542.523,E2 -31542.523} C_VEL
LIN {X 0,Y 210.584,Z 1005.565,A -85,B 0,C 180,E1 -31550.137,E2 -31550.137} C_VEL
LIN {X 0,Y 221.706,Z 1012.517,A -85,B 0,C 180,E1 -31555.505,E2 -31555.505} C_VEL
LIN {X 0,Y 231.438,Z 1018.838,A -85,B 0,C 180,E1 -31559.932,E2 -31559.932} C_VEL
LIN {X 0,Y 237.41,Z 1022.926,A -85,B 0,C 180,E1 -31562.632,E2 -31562.632} C_VEL
LIN {X 0,Y 243.356,Z 1027.109,A -85,B 0,C 180,E1 -31565.401,E2 -31565.401} C_VEL
LIN {X 0,Y 247.381,Z 1030.02,A -85,B 0,C 180,E1 -31567.413,E2 -31567.413} C_VEL
LIN {X 0,Y 252.858,Z 1033.9,A -85,B 0,C 180,E1 -31570.517,E2 -31570.517} C_VEL
LIN {X 0,Y 256.971,Z 1036.737,A -85,B 0,C 180,E1 -31573.179,E2 -31573.179} C_VEL
LIN {X 0,Y 259.271,Z 1038.411,A -85,B 0,C 180,E1 -31574.939,E2 -31574.939} C_VEL
LIN {X 0,Y 260.127,Z 1039.787,A -85,B 0,C 180,E1 -31576.196,E2 -31576.196} C_VEL
LIN {X 0,Y 259.74,Z 1042.262,A -85,B 0,C 180,E1 -31578.312,E2 -31578.312} C_VEL
LIN {X 0,Y 259.194,Z 1044.047,A -85,B 0,C 180,E1 -31580.037,E2 -31580.037} C_VEL
LIN {X 0,Y 259.473,Z 1044.975,A -85,B 0,C 180,E1 -31581.341,E2 -31581.341} C_VEL
LIN {X 0,Y 259.803,Z 1045.175,A -85,B 0,C 180,E1 -31581.772,E2 -31581.772} C_VEL
LIN {X 0,Y 261.547,Z 1045.975,A -85,B 0,C 180,E1 -31583.83,E2 -31583.83} C_VEL
LIN {X 0,Y 262.568,Z 1046.41,A -85,B 0,C 180,E1 -31585.394,E2 -31585.394} C_VEL
LIN {X 0,Y 263.269,Z 1046.709,A -85,B 0,C 180,E1 -31586.94,E2 -31586.94} C_VEL
LIN {X 0,Y 263.666,Z 1046.892,A -85,B 0,C 180,E1 -31588.473,E2 -31588.473} C_VEL
LIN {X 0,Y 263.868,Z 1046.932,A -85,B 0,C 180,E1 -31590,E2 -31590} C_VEL
LIN {X 0,Y 263.644,Z 1046.897,A -85,B 0,C 180,E1 -31591.527,E2 -31591.527} C_VEL
LIN {X 0,Y 263.221,Z 1046.721,A -85,B 0,C 180,E1 -31593.061,E2 -31593.061} C_VEL
LIN {X 0,Y 262.495,Z 1046.428,A -85,B 0,C 180,E1 -31594.607,E2 -31594.607} C_VEL
LIN {X 0,Y 261.5,Z 1045.991,A -85,B 0,C 180,E1 -31596.171,E2 -31596.171} C_VEL
LIN {X 0,Y 260.26,Z 1045.393,A -85,B 0,C 180,E1 -31597.759,E2 -31597.759} C_VEL
LIN {X 0,Y 257.452,Z 1043.939,A -85,B 0,C 180,E1 -31600.666,E2 -31600.666} C_VEL
LIN {X 0,Y 253.604,Z 1041.387,A -85,B 0,C 180,E1 -31604.088,E2 -31604.088} C_VEL
LIN {X 0,Y 249.801,Z 1038.668,A -85,B 0,C 180,E1 -31606.951,E2 -31606.951} C_VEL
LIN {X 0,Y 244.709,Z 1035.09,A -85,B 0,C 180,E1 -31610.159,E2 -31610.159} C_VEL
LIN {X 0,Y 237.986,Z 1030.336,A -85,B 0,C 180,E1 -31613.73,E2 -31613.73} C_VEL
LIN {X 0,Y 229.821,Z 1024.904,A -85,B 0,C 180,E1 -31617.524,E2 -31617.524} C_VEL
LIN {X 0,Y 224.355,Z 1021.361,A -85,B 0,C 180,E1 -31620.079,E2 -31620.079} C_VEL
LIN {X 0,Y 217.279,Z 1017.003,A -85,B 0,C 180,E1 -31623.357,E2 -31623.357} C_VEL
LIN {X 0,Y 209.417,Z 1012.283,A -85,B 0,C 180,E1 -31627.161,E2 -31627.161} C_VEL
LIN {X 0,Y 196.426,Z 1004.22,A -85,B 0,C 180,E1 -31634.31,E2 -31634.31} C_VEL
LIN {X 0,Y 183.399,Z 992.927,A -85,B 0,C 180,E1 -31644.914,E2 -31644.914} C_VEL
LIN {X 0,Y 177.705,Z 982.565,A -85,B 0,C 180,E1 -31654.213,E2 -31654.213} C_VEL
LIN {X 0,Y 176.655,Z 975.886,A -85,B 0,C 180,E1 -31659.757,E2 -31659.757} C_VEL
LIN {X 0,Y 175.552,Z 976.72,A -85,B 0,C 180,E1 -31660.18,E2 -31660.18} C_VEL
LIN {X 0,Y 165.082,Z 989.401,A -85,B 0,C 180,E1 -31659.484,E2 -31659.484} C_VEL
LIN {X 0,Y 154.28,Z 1000.586,A -85,B 0,C 180,E1 -31658.742,E2 -31658.742} C_VEL
LIN {X 0,Y 145.778,Z 1008.371,A -85,B 0,C 180,E1 -31658.128,E2 -31658.128} C_VEL
LIN {X 0,Y 133.633,Z 1018.148,A -85,B 0,C 180,E1 -31656.974,E2 -31656.974} C_VEL
LIN {X 0,Y 121.448,Z 1026.575,A -85,B 0,C 180,E1 -31655.697,E2 -31655.697} C_VEL
LIN {X 0,Y 109.315,Z 1033.792,A -85,B 0,C 180,E1 -31654.165,E2 -31654.165} C_VEL
LIN {X 0,Y 98.997,Z 1039.147,A -85,B 0,C 180,E1 -31652.545,E2 -31652.545} C_VEL
LIN {X 0,Y 88.784,Z 1043.788,A -85,B 0,C 180,E1 -31650.542,E2 -31650.542} C_VEL
LIN {X 0,Y 75.348,Z 1048.906,A -85,B 0,C 180,E1 -31647.082,E2 -31647.082} C_VEL
LIN {X 0,Y 62.327,Z 1052.92,A -85,B 0,C 180,E1 -31642.12,E2 -31642.12} C_VEL
LIN {X 0,Y 50.057,Z 1055.9,A -85,B 0,C 180,E1 -31634.586,E2 -31634.586} C_VEL
LIN {X 0,Y 44.389,Z 1057.099,A -85,B 0,C 180,E1 -31629.294,E2 -31629.294} C_VEL
LIN {X 0,Y 34.999,Z 1058.591,A -85,B 0,C 180,E1 -31613.678,E2 -31613.678} C_VEL
LIN {X 0,Y 30.037,Z 1059.136,A -85,B 0,C 180,E1 -31590,E2 -31590} C_VEL
LIN {X 0,Y 34.995,Z 1058.591,A -85,B 0,C 180,E1 -31566.319,E2 -31566.319} C_VEL
LIN {X 0,Y 44.373,Z 1057.099,A -85,B 0,C 180,E1 -31550.69,E2 -31550.69} C_VEL
LIN {X 0,Y 56.047,Z 1054.596,A -85,B 0,C 180,E1 -31541.206,E2 -31541.206} C_VEL
LIN {X 0,Y 72.042,Z 1049.998,A -85,B 0,C 180,E1 -31533.985,E2 -31533.985} C_VEL
LIN {X 0,Y 82.036,Z 1046.489,A -85,B 0,C 180,E1 -31531.055,E2 -31531.055} C_VEL
LIN {X 0,Y 95.576,Z 1040.77,A -85,B 0,C 180,E1 -31528.07,E2 -31528.07} C_VEL
LIN {X 0,Y 105.846,Z 1035.704,A -85,B 0,C 180,E1 -31526.317,E2 -31526.317} C_VEL
LIN {X 0,Y 119.365,Z 1027.906,A -85,B 0,C 180,E1 -31524.544,E2 -31524.544} C_VEL
LIN {X 0,Y 131.897,Z 1019.425,A -85,B 0,C 180,E1 -31523.202,E2 -31523.202} C_VEL
LIN {X 0,Y 140.613,Z 1012.755,A -85,B 0,C 180,E1 -31522.388,E2 -31522.388} C_VEL
LIN {X 0,Y 151.047,Z 1003.654,A -85,B 0,C 180,E1 -31521.48,E2 -31521.48} C_VEL
LIN {X 0,Y 161.576,Z 993.207,A -85,B 0,C 180,E1 -31520.748,E2 -31520.748} C_VEL
LIN {X 0,Y 171.205,Z 982.162,A -85,B 0,C 180,E1 -31520.117,E2 -31520.117} C_VEL
LIN {X 0,Y 175.066,Z 977.379,A -85,B 0,C 180,E1 -31519.889,E2 -31519.889} C_VEL
LIN {X 0,Y 176.628,Z 975.927,A -85,B 0,C 180,E1 -31520.248,E2 -31520.248} C_VEL
LIN {X 0,Y 179.16,Z 986.41,A -85,B 0,C 180,E1 -31529.101,E2 -31529.101} C_VEL
LIN {X 0,Y 187.854,Z 997.642,A -85,B 0,C 180,E1 -31539.493,E2 -31539.493} C_VEL
LIN {X 0,Y 200.845,Z 1007.108,A -85,B 0,C 180,E1 -31548.33,E2 -31548.33} C_VEL
LIN {X 0,Y 210.311,Z 1012.875,A -85,B 0,C 180,E1 -31553.321,E2 -31553.321} C_VEL
LIN {X 0,Y 219.906,Z 1018.594,A -85,B 0,C 180,E1 -31557.876,E2 -31557.876} C_VEL
LIN {X 0,Y 227.849,Z 1023.549,A -85,B 0,C 180,E1 -31561.53,E2 -31561.53} C_VEL
LIN {X 0,Y 233.879,Z 1027.564,A -85,B 0,C 180,E1 -31564.353,E2 -31564.353} C_VEL
LIN {X 0,Y 237.94,Z 1030.396,A -85,B 0,C 180,E1 -31566.295,E2 -31566.295} C_VEL
LIN {X 0,Y 241.94,Z 1033.17,A -85,B 0,C 180,E1 -31568.363,E2 -31568.363} C_VEL
LIN {X 0,Y 245.906,Z 1035.966,A -85,B 0,C 180,E1 -31570.583,E2 -31570.583} C_VEL
LIN {X 0,Y 250.777,Z 1039.374,A -85,B 0,C 180,E1 -31573.725,E2 -31573.725} C_VEL
LIN {X 0,Y 253.588,Z 1041.396,A -85,B 0,C 180,E1 -31575.926,E2 -31575.926} C_VEL
LIN {X 0,Y 257.451,Z 1043.94,A -85,B 0,C 180,E1 -31579.335,E2 -31579.335} C_VEL
LIN {X 0,Y 259.803,Z 1045.175,A -85,B 0,C 180,E1 -31581.772,E2 -31581.772} C_VEL
LIN {X 0,Y 260.286,Z 1045.902,A -85,B 0,C 180,E1 -31583.056,E2 -31583.056} C_VEL
LIN {X 0,Y 259.731,Z 1046.784,A -85,B 0,C 180,E1 -31584.346,E2 -31584.346} C_VEL
LIN {X 0,Y 257.008,Z 1048.699,A -85,B 0,C 180,E1 -31587.84,E2 -31587.84} C_VEL
LIN {X 0,Y 256.861,Z 1048.831,A -85,B 0,C 180,E1 -31588.738,E2 -31588.738} C_VEL
LIN {X 0,Y 257.048,Z 1048.861,A -85,B 0,C 180,E1 -31590,E2 -31590} C_VEL
LIN {X 0,Y 256.813,Z 1048.828,A -85,B 0,C 180,E1 -31591.568,E2 -31591.568} C_VEL
LIN {X 0,Y 256.317,Z 1048.661,A -85,B 0,C 180,E1 -31593.143,E2 -31593.143} C_VEL
LIN {X 0,Y 255.527,Z 1048.337,A -85,B 0,C 180,E1 -31594.733,E2 -31594.733} C_VEL
LIN {X 0,Y 254.436,Z 1047.848,A -85,B 0,C 180,E1 -31596.343,E2 -31596.343} C_VEL
LIN {X 0,Y 253.089,Z 1047.187,A -85,B 0,C 180,E1 -31597.981,E2 -31597.981} C_VEL
LIN {X 0,Y 250.361,Z 1045.712,A -85,B 0,C 180,E1 -31600.739,E2 -31600.739} C_VEL
LIN {X 0,Y 246.439,Z 1043.043,A -85,B 0,C 180,E1 -31604.163,E2 -31604.163} C_VEL
LIN {X 0,Y 242.539,Z 1040.362,A -85,B 0,C 180,E1 -31607.017,E2 -31607.017} C_VEL
LIN {X 0,Y 238.568,Z 1037.484,A -85,B 0,C 180,E1 -31609.494,E2 -31609.494} C_VEL
LIN {X 0,Y 234.524,Z 1034.717,A -85,B 0,C 180,E1 -31611.726,E2 -31611.726} C_VEL
LIN {X 0,Y 230.433,Z 1031.919,A -85,B 0,C 180,E1 -31613.8,E2 -31613.8} C_VEL
LIN {X 0,Y 222.241,Z 1026.848,A -85,B 0,C 180,E1 -31617.694,E2 -31617.694} C_VEL
LIN {X 0,Y 213.62,Z 1021.724,A -85,B 0,C 180,E1 -31621.761,E2 -31621.761} C_VEL
LIN {X 0,Y 206.101,Z 1017.389,A -85,B 0,C 180,E1 -31625.428,E2 -31625.428} C_VEL
LIN {X 0,Y 193.911,Z 1010.325,A -85,B 0,C 180,E1 -31632.015,E2 -31632.015} C_VEL
LIN {X 0,Y 181.029,Z 1000.783,A -85,B 0,C 180,E1 -31641.6,E2 -31641.6} C_VEL
LIN {X 0,Y 174.012,Z 991.242,A -85,B 0,C 180,E1 -31651.011,E2 -31651.011} C_VEL
LIN {X 0,Y 172.114,Z 984.435,A -85,B 0,C 180,E1 -31657.264,E2 -31657.264} C_VEL
LIN {X 0,Y 170.223,Z 986.352,A -85,B 0,C 180,E1 -31657.403,E2 -31657.403} C_VEL
LIN {X 0,Y 159.242,Z 998.223,A -85,B 0,C 180,E1 -31656.51,E2 -31656.51} C_VEL
LIN {X 0,Y 148.589,Z 1008.168,A -85,B 0,C 180,E1 -31655.57,E2 -31655.57} C_VEL
LIN {X 0,Y 136.597,Z 1017.943,A -85,B 0,C 180,E1 -31654.205,E2 -31654.205} C_VEL
LIN {X 0,Y 124.584,Z 1026.37,A -85,B 0,C 180,E1 -31652.679,E2 -31652.679} C_VEL
LIN {X 0,Y 112.643,Z 1033.586,A -85,B 0,C 180,E1 -31650.864,E2 -31650.864} C_VEL
LIN {X 0,Y 102.522,Z 1038.942,A -85,B 0,C 180,E1 -31648.967,E2 -31648.967} C_VEL
LIN {X 0,Y 89.257,Z 1044.931,A -85,B 0,C 180,E1 -31645.765,E2 -31645.765} C_VEL
LIN {X 0,Y 76.315,Z 1049.792,A -85,B 0,C 180,E1 -31641.514,E2 -31641.514} C_VEL
LIN {X 0,Y 61.045,Z 1054.386,A -85,B 0,C 180,E1 -31633.689,E2 -31633.689} C_VEL
LIN {X 0,Y 50.181,Z 1056.89,A -85,B 0,C 180,E1 -31624.069,E2 -31624.069} C_VEL
LIN {X 0,Y 41.667,Z 1058.382,A -85,B 0,C 180,E1 -31609.714,E2 -31609.714} C_VEL
LIN {X 0,Y 37.174,Z 1058.929,A -85,B 0,C 180,E1 -31590,E2 -31590} C_VEL
LIN {X 0,Y 41.662,Z 1058.382,A -85,B 0,C 180,E1 -31570.283,E2 -31570.283} C_VEL
LIN {X 0,Y 52.639,Z 1056.316,A -85,B 0,C 180,E1 -31553.23,E2 -31553.23} C_VEL
LIN {X 0,Y 61.04,Z 1054.387,A -85,B 0,C 180,E1 -31546.306,E2 -31546.306} C_VEL
LIN {X 0,Y 76.323,Z 1049.792,A -85,B 0,C 180,E1 -31538.494,E2 -31538.494} C_VEL
LIN {X 0,Y 89.22,Z 1044.933,A -85,B 0,C 180,E1 -31534.2,E2 -31534.2} C_VEL
LIN {X 0,Y 102.516,Z 1038.943,A -85,B 0,C 180,E1 -31531.028,E2 -31531.028} C_VEL
LIN {X 0,Y 116.024,Z 1031.674,A -85,B 0,C 180,E1 -31528.563,E2 -31528.563} C_VEL
LIN {X 0,Y 131.444,Z 1021.778,A -85,B 0,C 180,E1 -31526.42,E2 -31526.42} C_VEL
LIN {X 0,Y 143.483,Z 1012.552,A -85,B 0,C 180,E1 -31525.024,E2 -31525.024} C_VEL
LIN {X 0,Y 153.825,Z 1003.449,A -85,B 0,C 180,E1 -31523.972,E2 -31523.972} C_VEL
LIN {X 0,Y 164.245,Z 993.005,A -85,B 0,C 180,E1 -31523.081,E2 -31523.081} C_VEL
LIN {X 0,Y 170.2,Z 986.363,A -85,B 0,C 180,E1 -31522.586,E2 -31522.586} C_VEL
LIN {X 0,Y 172.096,Z 984.445,A -85,B 0,C 180,E1 -31522.729,E2 -31522.729} C_VEL
LIN {X 0,Y 175.352,Z 993.754,A -85,B 0,C 180,E1 -31531.401,E2 -31531.401} C_VEL
LIN {X 0,Y 184.808,Z 1004.092,A -85,B 0,C 180,E1 -31541.72,E2 -31541.72} C_VEL
LIN {X 0,Y 199.116,Z 1013.396,A -85,B 0,C 180,E1 -31550.941,E2 -31550.941} C_VEL
LIN {X 0,Y 210.297,Z 1019.816,A -85,B 0,C 180,E1 -31556.665,E2 -31556.665} C_VEL
LIN {X 0,Y 218.193,Z 1024.4,A -85,B 0,C 180,E1 -31560.419,E2 -31560.419} C_VEL
LIN {X 0,Y 224.244,Z 1028.059,A -85,B 0,C 180,E1 -31563.265,E2 -31563.265} C_VEL
LIN {X 0,Y 231.484,Z 1032.659,A -85,B 0,C 180,E1 -31566.754,E2 -31566.754} C_VEL
LIN {X 0,Y 235.894,Z 1035.709,A -85,B 0,C 180,E1 -31569.053,E2 -31569.053} C_VEL
LIN {X 0,Y 239.653,Z 1038.307,A -85,B 0,C 180,E1 -31571.181,E2 -31571.181} C_VEL
LIN {X 0,Y 242.797,Z 1040.571,A -85,B 0,C 180,E1 -31573.175,E2 -31573.175} C_VEL
LIN {X 0,Y 246.427,Z 1043.033,A -85,B 0,C 180,E1 -31575.848,E2 -31575.848} C_VEL
LIN {X 0,Y 249.675,Z 1045.332,A -85,B 0,C 180,E1 -31578.636,E2 -31578.636} C_VEL
LIN {X 0,Y 251.508,Z 1046.349,A -85,B 0,C 180,E1 -31580.348,E2 -31580.348} C_VEL
LIN {X 0,Y 253.084,Z 1047.185,A -85,B 0,C 180,E1 -31582.019,E2 -31582.019} C_VEL
LIN {X 0,Y 254.535,Z 1047.855,A -85,B 0,C 180,E1 -31583.713,E2 -31583.713} C_VEL
LIN {X 0,Y 255.602,Z 1048.322,A -85,B 0,C 180,E1 -31585.269,E2 -31585.269} C_VEL
LIN {X 0,Y 256.393,Z 1048.644,A -85,B 0,C 180,E1 -31586.857,E2 -31586.857} C_VEL
LIN {X 0,Y 256.861,Z 1048.831,A -85,B 0,C 180,E1 -31588.738,E2 -31588.738} C_VEL
LIN {X 0,Y 256.238,Z 1049.095,A -85,B 0,C 180,E1 -31590.047,E2 -31590.047} C_VEL
LIN {X 0,Y 254.538,Z 1049.413,A -85,B 0,C 180,E1 -31591.324,E2 -31591.324} C_VEL
LIN {X 0,Y 248.756,Z 1049.865,A -85,B 0,C 180,E1 -31594.757,E2 -31594.757} C_VEL
LIN {X 0,Y 247.881,Z 1049.638,A -85,B 0,C 180,E1 -31595.666,E2 -31595.666} C_VEL
LIN {X 0,Y 245.806,Z 1048.582,A -85,B 0,C 180,E1 -31598.219,E2 -31598.219} C_VEL
LIN {X 0,Y 243.219,Z 1047.106,A -85,B 0,C 180,E1 -31600.753,E2 -31600.753} C_VEL
LIN {X 0,Y 239.22,Z 1044.475,A -85,B 0,C 180,E1 -31604.19,E2 -31604.19} C_VEL
LIN {X 0,Y 234.567,Z 1041.197,A -85,B 0,C 180,E1 -31607.434,E2 -31607.434} C_VEL
LIN {X 0,Y 231.054,Z 1038.795,A -85,B 0,C 180,E1 -31609.547,E2 -31609.547} C_VEL
LIN {X 0,Y 224.884,Z 1034.753,A -85,B 0,C 180,E1 -31612.868,E2 -31612.868} C_VEL
LIN {X 0,Y 216.167,Z 1029.641,A -85,B 0,C 180,E1 -31617.075,E2 -31617.075} C_VEL
LIN {X 0,Y 209.675,Z 1026.036,A -85,B 0,C 180,E1 -31620.183,E2 -31620.183} C_VEL
LIN {X 0,Y 202.498,Z 1022.104,A -85,B 0,C 180,E1 -31623.731,E2 -31623.731} C_VEL
LIN {X 0,Y 191.467,Z 1016.157,A -85,B 0,C 180,E1 -31629.573,E2 -31629.573} C_VEL
LIN {X 0,Y 178.761,Z 1007.993,A -85,B 0,C 180,E1 -31638.328,E2 -31638.328} C_VEL
LIN {X 0,Y 169.849,Z 998.169,A -85,B 0,C 180,E1 -31648.855,E2 -31648.855} C_VEL
LIN {X 0,Y 167.631,Z 992.646,A -85,B 0,C 180,E1 -31654.438,E2 -31654.438} C_VEL
LIN {X 0,Y 166.118,Z 993.984,A -85,B 0,C 180,E1 -31654.557,E2 -31654.557} C_VEL
LIN {X 0,Y 155.114,Z 1004.906,A -85,B 0,C 180,E1 -31653.486,E2 -31653.486} C_VEL
LIN {X 0,Y 141.571,Z 1016.455,A -85,B 0,C 180,E1 -31651.78,E2 -31651.78} C_VEL
LIN {X 0,Y 129.729,Z 1025.055,A -85,B 0,C 180,E1 -31650.086,E2 -31650.086} C_VEL
LIN {X 0,Y 119.299,Z 1031.665,A -85,B 0,C 180,E1 -31648.337,E2 -31648.337} C_VEL
LIN {X 0,Y 106.407,Z 1038.738,A -85,B 0,C 180,E1 -31645.648,E2 -31645.648} C_VEL
LIN {X 0,Y 93.498,Z 1044.725,A -85,B 0,C 180,E1 -31642.114,E2 -31642.114} C_VEL
LIN {X 0,Y 84.052,Z 1048.495,A -85,B 0,C 180,E1 -31638.809,E2 -31638.809} C_VEL
LIN {X 0,Y 72.105,Z 1052.508,A -85,B 0,C 180,E1 -31633.021,E2 -31633.021} C_VEL
LIN {X 0,Y 61.163,Z 1055.487,A -85,B 0,C 180,E1 -31625.066,E2 -31625.066} C_VEL
LIN {X 0,Y 52.026,Z 1057.484,A -85,B 0,C 180,E1 -31613.907,E2 -31613.907} C_VEL
LIN {X 0,Y 45.85,Z 1058.494,A -85,B 0,C 180,E1 -31598.817,E2 -31598.817} C_VEL
LIN {X 0,Y 44.334,Z 1058.722,A -85,B 0,C 180,E1 -31590,E2 -31590} C_VEL
LIN {X 0,Y 48.47,Z 1058.173,A -85,B 0,C 180,E1 -31573.143,E2 -31573.143} C_VEL
LIN {X 0,Y 57.916,Z 1056.272,A -85,B 0,C 180,E1 -31558.146,E2 -31558.146} C_VEL
LIN {X 0,Y 66.452,Z 1054.177,A -85,B 0,C 180,E1 -31550.614,E2 -31550.614} C_VEL
LIN {X 0,Y 81.017,Z 1049.586,A -85,B 0,C 180,E1 -31542.496,E2 -31542.496} C_VEL
LIN {X 0,Y 90.315,Z 1046.075,A -85,B 0,C 180,E1 -31538.909,E2 -31538.909} C_VEL
LIN {X 0,Y 103.135,Z 1040.36,A -85,B 0,C 180,E1 -31535.145,E2 -31535.145} C_VEL
LIN {X 0,Y 116.311,Z 1033.381,A -85,B 0,C 180,E1 -31532.23,E2 -31532.23} C_VEL
LIN {X 0,Y 128.049,Z 1026.165,A -85,B 0,C 180,E1 -31530.183,E2 -31530.183} C_VEL
LIN {X 0,Y 139.893,Z 1017.737,A -85,B 0,C 180,E1 -31528.461,E2 -31528.461} C_VEL
LIN {X 0,Y 151.705,Z 1007.964,A -85,B 0,C 180,E1 -31526.904,E2 -31526.904} C_VEL
LIN {X 0,Y 163.744,Z 996.518,A -85,B 0,C 180,E1 -31525.669,E2 -31525.669} C_VEL
LIN {X 0,Y 166.106,Z 993.993,A -85,B 0,C 180,E1 -31525.442,E2 -31525.442} C_VEL
LIN {X 0,Y 167.605,Z 992.669,A -85,B 0,C 180,E1 -31525.56,E2 -31525.56} C_VEL
LIN {X 0,Y 172.242,Z 1001.654,A -85,B 0,C 180,E1 -31534.836,E2 -31534.836} C_VEL
LIN {X 0,Y 181.827,Z 1010.177,A -85,B 0,C 180,E1 -31544.085,E2 -31544.085} C_VEL
LIN {X 0,Y 195.085,Z 1018.134,A -85,B 0,C 180,E1 -31552.424,E2 -31552.424} C_VEL
LIN {X 0,Y 204.56,Z 1023.252,A -85,B 0,C 180,E1 -31557.323,E2 -31557.323} C_VEL
LIN {X 0,Y 212.546,Z 1027.621,A -85,B 0,C 180,E1 -31561.191,E2 -31561.191} C_VEL
LIN {X 0,Y 218.687,Z 1031.137,A -85,B 0,C 180,E1 -31564.135,E2 -31564.135} C_VEL
LIN {X 0,Y 224.826,Z 1034.775,A -85,B 0,C 180,E1 -31567.138,E2 -31567.138} C_VEL
LIN {X 0,Y 231.109,Z 1038.864,A -85,B 0,C 180,E1 -31570.509,E2 -31570.509} C_VEL
LIN {X 0,Y 235.197,Z 1041.649,A -85,B 0,C 180,E1 -31572.977,E2 -31572.977} C_VEL
LIN {X 0,Y 240.041,Z 1045.08,A -85,B 0,C 180,E1 -31576.454,E2 -31576.454} C_VEL
LIN {X 0,Y 244.104,Z 1047.625,A -85,B 0,C 180,E1 -31580.053,E2 -31580.053} C_VEL
LIN {X 0,Y 245.803,Z 1048.584,A -85,B 0,C 180,E1 -31581.781,E2 -31581.781} C_VEL
LIN {X 0,Y 247.477,Z 1049.433,A -85,B 0,C 180,E1 -31583.687,E2 -31583.687} C_VEL
LIN {X 0,Y 248.522,Z 1049.87,A -85,B 0,C 180,E1 -31585.133,E2 -31585.133} C_VEL
LIN {X 0,Y 249.388,Z 1050.198,A -85,B 0,C 180,E1 -31586.769,E2 -31586.769} C_VEL
LIN {X 0,Y 249.937,Z 1050.405,A -85,B 0,C 180,E1 -31588.773,E2 -31588.773} C_VEL
LIN {X 0,Y 250.125,Z 1050.446,A -85,B 0,C 180,E1 -31590,E2 -31590} C_VEL
LIN {X 0,Y 249.854,Z 1050.403,A -85,B 0,C 180,E1 -31591.612,E2 -31591.612} C_VEL
LIN {X 0,Y 249.319,Z 1050.212,A -85,B 0,C 180,E1 -31593.232,E2 -31593.232} C_VEL
LIN {X 0,Y 247.881,Z 1049.638,A -85,B 0,C 180,E1 -31595.666,E2 -31595.666} C_VEL
LIN {X 0,Y 246.245,Z 1049.293,A -85,B 0,C 180,E1 -31596.975,E2 -31596.975} C_VEL
LIN {X 0,Y 243.59,Z 1049.015,A -85,B 0,C 180,E1 -31598.217,E2 -31598.217} C_VEL
LIN {X 0,Y 237.308,Z 1048.175,A -85,B 0,C 180,E1 -31600.664,E2 -31600.664} C_VEL
LIN {X 0,Y 234.702,Z 1047.347,A -85,B 0,C 180,E1 -31601.97,E2 -31601.97} C_VEL
LIN {X 0,Y 234.05,Z 1046.974,A -85,B 0,C 180,E1 -31602.426,E2 -31602.426} C_VEL
LIN {X 0,Y 231.931,Z 1045.505,A -85,B 0,C 180,E1 -31604.152,E2 -31604.152} C_VEL
LIN {X 0,Y 227.838,Z 1042.689,A -85,B 0,C 180,E1 -31607.016,E2 -31607.016} C_VEL
LIN {X 0,Y 223.652,Z 1040.007,A -85,B 0,C 180,E1 -31609.49,E2 -31609.49} C_VEL
LIN {X 0,Y 219.463,Z 1037.47,A -85,B 0,C 180,E1 -31611.772,E2 -31611.772} C_VEL
LIN {X 0,Y 215.228,Z 1035.15,A -85,B 0,C 180,E1 -31613.895,E2 -31613.895} C_VEL
LIN {X 0,Y 206.891,Z 1030.66,A -85,B 0,C 180,E1 -31617.97,E2 -31617.97} C_VEL
LIN {X 0,Y 198.624,Z 1026.411,A -85,B 0,C 180,E1 -31622.055,E2 -31622.055} C_VEL
LIN {X 0,Y 187.372,Z 1020.718,A -85,B 0,C 180,E1 -31628.033,E2 -31628.033} C_VEL
LIN {X 0,Y 174.494,Z 1013.133,A -85,B 0,C 180,E1 -31636.789,E2 -31636.789} C_VEL
LIN {X 0,Y 165.69,Z 1004.766,A -85,B 0,C 180,E1 -31646.537,E2 -31646.537} C_VEL
LIN {X 0,Y 164.246,Z 1002.463,A -85,B 0,C 180,E1 -31649.106,E2 -31649.106} C_VEL
LIN {X 0,Y 162.548,Z 1000.729,A -85,B 0,C 180,E1 -31651.602,E2 -31651.602} C_VEL
LIN {X 0,Y 153.378,Z 1009.225,A -85,B 0,C 180,E1 -31650.526,E2 -31650.526} C_VEL
LIN {X 0,Y 143.434,Z 1017.534,A -85,B 0,C 180,E1 -31649.031,E2 -31649.031} C_VEL
LIN {X 0,Y 131.803,Z 1025.961,A -85,B 0,C 180,E1 -31647.119,E2 -31647.119} C_VEL
LIN {X 0,Y 120.308,Z 1033.175,A -85,B 0,C 180,E1 -31644.866,E2 -31644.866} C_VEL
LIN {X 0,Y 107.457,Z 1040.154,A -85,B 0,C 180,E1 -31641.704,E2 -31641.704} C_VEL
LIN {X 0,Y 95.032,Z 1045.867,A -85,B 0,C 180,E1 -31637.691,E2 -31637.691} C_VEL
LIN {X 0,Y 83.123,Z 1050.473,A -85,B 0,C 180,E1 -31632.561,E2 -31632.561} C_VEL
LIN {X 0,Y 72.175,Z 1053.968,A -85,B 0,C 180,E1 -31625.749,E2 -31625.749} C_VEL
LIN {X 0,Y 62.637,Z 1056.473,A -85,B 0,C 180,E1 -31616.666,E2 -31616.666} C_VEL
LIN {X 0,Y 55.402,Z 1057.964,A -85,B 0,C 180,E1 -31604.697,E2 -31604.697} C_VEL
LIN {X 0,Y 51.484,Z 1058.515,A -85,B 0,C 180,E1 -31590,E2 -31590} C_VEL
LIN {X 0,Y 55.394,Z 1057.964,A -85,B 0,C 180,E1 -31575.301,E2 -31575.301} C_VEL
LIN {X 0,Y 63.556,Z 1056.224,A -85,B 0,C 180,E1 -31562.203,E2 -31562.203} C_VEL
LIN {X 0,Y 72.167,Z 1053.968,A -85,B 0,C 180,E1 -31554.247,E2 -31554.247} C_VEL
LIN {X 0,Y 86.048,Z 1049.381,A -85,B 0,C 180,E1 -31546.035,E2 -31546.035} C_VEL
LIN {X 0,Y 98.053,Z 1044.52,A -85,B 0,C 180,E1 -31541.187,E2 -31541.187} C_VEL
LIN {X 0,Y 110.613,Z 1038.533,A -85,B 0,C 180,E1 -31537.421,E2 -31537.421} C_VEL
LIN {X 0,Y 125.353,Z 1030.213,A -85,B 0,C 180,E1 -31534.1,E2 -31534.1} C_VEL
LIN {X 0,Y 138.448,Z 1021.367,A -85,B 0,C 180,E1 -31531.761,E2 -31531.761} C_VEL
LIN {X 0,Y 150.076,Z 1012.147,A -85,B 0,C 180,E1 -31529.966,E2 -31529.966} C_VEL
LIN {X 0,Y 160.227,Z 1003.039,A -85,B 0,C 180,E1 -31528.69,E2 -31528.69} C_VEL
LIN {X 0,Y 162.134,Z 1001.173,A -85,B 0,C 180,E1 -31528.477,E2 -31528.477} C_VEL
LIN {X 0,Y 164.436,Z 1002.799,A -85,B 0,C 180,E1 -31531.265,E2 -31531.265} C_VEL
LIN {X 0,Y 171.833,Z 1011.125,A -85,B 0,C 180,E1 -31540.873,E2 -31540.873} C_VEL
LIN {X 0,Y 183.874,Z 1018.837,A -85,B 0,C 180,E1 -31549.855,E2 -31549.855} C_VEL
LIN {X 0,Y 191.091,Z 1022.59,A -85,B 0,C 180,E1 -31554.009,E2 -31554.009} C_VEL
LIN {X 0,Y 200.796,Z 1027.546,A -85,B 0,C 180,E1 -31559.037,E2 -31559.037} C_VEL
LIN {X 0,Y 208.963,Z 1031.769,A -85,B 0,C 180,E1 -31563.031,E2 -31563.031} C_VEL
LIN {X 0,Y 217.343,Z 1036.306,A -85,B 0,C 180,E1 -31567.169,E2 -31567.169} C_VEL
LIN {X 0,Y 223.627,Z 1040.035,A -85,B 0,C 180,E1 -31570.528,E2 -31570.528} C_VEL
LIN {X 0,Y 227.83,Z 1042.697,A -85,B 0,C 180,E1 -31572.991,E2 -31572.991} C_VEL
LIN {X 0,Y 232.11,Z 1045.62,A -85,B 0,C 180,E1 -31575.982,E2 -31575.982} C_VEL
LIN {X 0,Y 236.038,Z 1048.265,A -85,B 0,C 180,E1 -31579.283,E2 -31579.283} C_VEL
LIN {X 0,Y 238.403,Z 1049.669,A -85,B 0,C 180,E1 -31581.524,E2 -31581.524} C_VEL
LIN {X 0,Y 240.39,Z 1050.591,A -85,B 0,C 180,E1 -31583.721,E2 -31583.721} C_VEL
LIN {X 0,Y 242.298,Z 1051.368,A -85,B 0,C 180,E1 -31586.674,E2 -31586.674} C_VEL
LIN {X 0,Y 242.874,Z 1051.604,A -85,B 0,C 180,E1 -31588.342,E2 -31588.342} C_VEL
LIN {X 0,Y 243.138,Z 1051.672,A -85,B 0,C 180,E1 -31590,E2 -31590} C_VEL
LIN {X 0,Y 242.828,Z 1051.613,A -85,B 0,C 180,E1 -31591.658,E2 -31591.658} C_VEL
LIN {X 0,Y 242.233,Z 1051.382,A -85,B 0,C 180,E1 -31593.326,E2 -31593.326} C_VEL
LIN {X 0,Y 240.385,Z 1050.599,A -85,B 0,C 180,E1 -31596.268,E2 -31596.268} C_VEL
LIN {X 0,Y 238.405,Z 1049.667,A -85,B 0,C 180,E1 -31598.476,E2 -31598.476} C_VEL
LIN {X 0,Y 236.039,Z 1048.263,A -85,B 0,C 180,E1 -31600.719,E2 -31600.719} C_VEL
LIN {X 0,Y 234.05,Z 1046.974,A -85,B 0,C 180,E1 -31602.426,E2 -31602.426} C_VEL
LIN {X 0,Y 231.691,Z 1045.977,A -85,B 0,C 180,E1 -31603.732,E2 -31603.732} C_VEL
LIN {X 0,Y 228.432,Z 1045.088,A -85,B 0,C 180,E1 -31604.951,E2 -31604.951} C_VEL
LIN {X 0,Y 218.759,Z 1042.465,A -85,B 0,C 180,E1 -31608.185,E2 -31608.185} C_VEL
LIN {X 0,Y 216.838,Z 1041.579,A -85,B 0,C 180,E1 -31609.087,E2 -31609.087} C_VEL
LIN {X 0,Y 211.878,Z 1038.906,A -85,B 0,C 180,E1 -31611.76,E2 -31611.76} C_VEL
LIN {X 0,Y 203.339,Z 1034.581,A -85,B 0,C 180,E1 -31616.023,E2 -31616.023} C_VEL
LIN {X 0,Y 194.605,Z 1030.349,A -85,B 0,C 180,E1 -31620.37,E2 -31620.37} C_VEL
LIN {X 0,Y 187.006,Z 1026.814,A -85,B 0,C 180,E1 -31624.313,E2 -31624.313} C_VEL
LIN {X 0,Y 176.212,Z 1021.436,A -85,B 0,C 180,E1 -31630.732,E2 -31630.732} C_VEL
LIN {X 0,Y 162.557,Z 1011.962,A -85,B 0,C 180,E1 -31642.752,E2 -31642.752} C_VEL
LIN {X 0,Y 159.198,Z 1007.734,A -85,B 0,C 180,E1 -31648.012,E2 -31648.012} C_VEL
LIN {X 0,Y 157.015,Z 1009.022,A -85,B 0,C 180,E1 -31648.257,E2 -31648.257} C_VEL
LIN {X 0,Y 147.252,Z 1017.329,A -85,B 0,C 180,E1 -31646.638,E2 -31646.638} C_VEL
LIN {X 0,Y 135.842,Z 1025.756,A -85,B 0,C 180,E1 -31644.57,E2 -31644.57} C_VEL
LIN {X 0,Y 124.582,Z 1032.969,A -85,B 0,C 180,E1 -31642.163,E2 -31642.163} C_VEL
LIN {X 0,Y 112.064,Z 1039.949,A -85,B 0,C 180,E1 -31638.812,E2 -31638.812} C_VEL
LIN {X 0,Y 100.017,Z 1045.66,A -85,B 0,C 180,E1 -31634.641,E2 -31634.641} C_VEL
LIN {X 0,Y 88.585,Z 1050.265,A -85,B 0,C 180,E1 -31629.396,E2 -31629.396} C_VEL
LIN {X 0,Y 78.157,Z 1053.758,A -85,B 0,C 180,E1 -31622.651,E2 -31622.651} C_VEL
LIN {X 0,Y 69.134,Z 1056.264,A -85,B 0,C 180,E1 -31613.993,E2 -31613.993} C_VEL
LIN {X 0,Y 62.381,Z 1057.754,A -85,B 0,C 180,E1 -31603.022,E2 -31603.022} C_VEL
LIN {X 0,Y 58.627,Z 1058.308,A -85,B 0,C 180,E1 -31590,E2 -31590} C_VEL
LIN {X 0,Y 62.372,Z 1057.754,A -85,B 0,C 180,E1 -31576.976,E2 -31576.976} C_VEL
LIN {X 0,Y 69.426,Z 1056.189,A -85,B 0,C 180,E1 -31565.648,E2 -31565.648} C_VEL
LIN {X 0,Y 78.148,Z 1053.759,A -85,B 0,C 180,E1 -31557.345,E2 -31557.345} C_VEL
LIN {X 0,Y 91.368,Z 1049.175,A -85,B 0,C 180,E1 -31549.171,E2 -31549.171} C_VEL
LIN {X 0,Y 102.949,Z 1044.313,A -85,B 0,C 180,E1 -31544.211,E2 -31544.211} C_VEL
LIN {X 0,Y 115.141,Z 1038.328,A -85,B 0,C 180,E1 -31540.274,E2 -31540.274} C_VEL
LIN {X 0,Y 128.662,Z 1030.53,A -85,B 0,C 180,E1 -31536.93,E2 -31536.93} C_VEL
LIN {X 0,Y 142.361,Z 1021.16,A -85,B 0,C 180,E1 -31534.22,E2 -31534.22} C_VEL
LIN {X 0,Y 153.772,Z 1011.941,A -85,B 0,C 180,E1 -31532.274,E2 -31532.274} C_VEL
LIN {X 0,Y 157.042,Z 1009.02,A -85,B 0,C 180,E1 -31531.759,E2 -31531.759} C_VEL
LIN {X 0,Y 159.18,Z 1007.751,A -85,B 0,C 180,E1 -31531.992,E2 -31531.992} C_VEL
LIN {X 0,Y 167.174,Z 1015.903,A -85,B 0,C 180,E1 -31542.27,E2 -31542.27} C_VEL
LIN {X 0,Y 179.672,Z 1023.227,A -85,B 0,C 180,E1 -31551.471,E2 -31551.471} C_VEL
LIN {X 0,Y 190.992,Z 1028.706,A -85,B 0,C 180,E1 -31557.814,E2 -31557.814} C_VEL
LIN {X 0,Y 199.149,Z 1032.568,A -85,B 0,C 180,E1 -31561.913,E2 -31561.913} C_VEL
LIN {X 0,Y 205.364,Z 1035.607,A -85,B 0,C 180,E1 -31564.984,E2 -31564.984} C_VEL
LIN {X 0,Y 212.688,Z 1039.357,A -85,B 0,C 180,E1 -31568.687,E2 -31568.687} C_VEL
LIN {X 0,Y 217.127,Z 1041.801,A -85,B 0,C 180,E1 -31571.115,E2 -31571.115} C_VEL
LIN {X 0,Y 220.954,Z 1043.979,A -85,B 0,C 180,E1 -31573.366,E2 -31573.366} C_VEL
LIN {X 0,Y 224.607,Z 1046.349,A -85,B 0,C 180,E1 -31575.926,E2 -31575.926} C_VEL
LIN {X 0,Y 226.58,Z 1047.693,A -85,B 0,C 180,E1 -31577.46,E2 -31577.46} C_VEL
LIN {X 0,Y 228.851,Z 1049.109,A -85,B 0,C 180,E1 -31579.382,E2 -31579.382} C_VEL
LIN {X 0,Y 230.846,Z 1050.225,A -85,B 0,C 180,E1 -31581.244,E2 -31581.244} C_VEL
LIN {X 0,Y 233.275,Z 1051.474,A -85,B 0,C 180,E1 -31583.821,E2 -31583.821} C_VEL
LIN {X 0,Y 235.129,Z 1052.329,A -85,B 0,C 180,E1 -31586.573,E2 -31586.573} C_VEL
LIN {X 0,Y 235.815,Z 1052.612,A -85,B 0,C 180,E1 -31588.292,E2 -31588.292} C_VEL
LIN {X 0,Y 236.104,Z 1052.693,A -85,B 0,C 180,E1 -31590,E2 -31590} C_VEL
LIN {X 0,Y 235.772,Z 1052.615,A -85,B 0,C 180,E1 -31591.708,E2 -31591.708} C_VEL
LIN {X 0,Y 235.064,Z 1052.332,A -85,B 0,C 180,E1 -31593.428,E2 -31593.428} C_VEL
LIN {X 0,Y 233.271,Z 1051.48,A -85,B 0,C 180,E1 -31596.168,E2 -31596.168} C_VEL
LIN {X 0,Y 230.847,Z 1050.225,A -85,B 0,C 180,E1 -31598.755,E2 -31598.755} C_VEL
LIN {X 0,Y 228.827,Z 1049.092,A -85,B 0,C 180,E1 -31600.641,E2 -31600.641} C_VEL
LIN {X 0,Y 226.605,Z 1047.692,A -85,B 0,C 180,E1 -31602.538,E2 -31602.538} C_VEL
LIN {X 0,Y 223.968,Z 1045.942,A -85,B 0,C 180,E1 -31604.538,E2 -31604.538} C_VEL
LIN {X 0,Y 220.429,Z 1043.658,A -85,B 0,C 180,E1 -31606.965,E2 -31606.965} C_VEL
LIN {X 0,Y 216.838,Z 1041.579,A -85,B 0,C 180,E1 -31609.087,E2 -31609.087} C_VEL
LIN {X 0,Y 213.731,Z 1040.387,A -85,B 0,C 180,E1 -31610.379,E2 -31610.379} C_VEL
LIN {X 0,Y 209.788,Z 1039.531,A -85,B 0,C 180,E1 -31611.558,E2 -31611.558} C_VEL
LIN {X 0,Y 201.21,Z 1038.053,A -85,B 0,C 180,E1 -31613.877,E2 -31613.877} C_VEL
LIN {X 0,Y 197.449,Z 1037.06,A -85,B 0,C 180,E1 -31615.195,E2 -31615.195} C_VEL
LIN {X 0,Y 196.397,Z 1036.648,A -85,B 0,C 180,E1 -31615.677,E2 -31615.677} C_VEL
LIN {X 0,Y 187.246,Z 1032.607,A -85,B 0,C 180,E1 -31620.316,E2 -31620.316} C_VEL
LIN {X 0,Y 175.486,Z 1027.429,A -85,B 0,C 180,E1 -31626.778,E2 -31626.778} C_VEL
LIN {X 0,Y 162.458,Z 1020.533,A -85,B 0,C 180,E1 -31636.2,E2 -31636.2} C_VEL
LIN {X 0,Y 155.358,Z 1014.496,A -85,B 0,C 180,E1 -31644.514,E2 -31644.514} C_VEL
LIN {X 0,Y 154.498,Z 1014.539,A -85,B 0,C 180,E1 -31644.963,E2 -31644.963} C_VEL
LIN {X 0,Y 141.703,Z 1024.442,A -85,B 0,C 180,E1 -31642.516,E2 -31642.516} C_VEL
LIN {X 0,Y 132.32,Z 1030.81,A -85,B 0,C 180,E1 -31640.406,E2 -31640.406} C_VEL
LIN {X 0,Y 119.926,Z 1038.123,A -85,B 0,C 180,E1 -31637.098,E2 -31637.098} C_VEL
LIN {X 0,Y 108.122,Z 1044.105,A -85,B 0,C 180,E1 -31633.038,E2 -31633.038} C_VEL
LIN {X 0,Y 96.928,Z 1048.97,A -85,B 0,C 180,E1 -31628.046,E2 -31628.046} C_VEL
LIN {X 0,Y 84.322,Z 1053.549,A -85,B 0,C 180,E1 -31620.005,E2 -31620.005} C_VEL
LIN {X 0,Y 75.539,Z 1056.109,A -85,B 0,C 180,E1 -31611.51,E2 -31611.51} C_VEL
LIN {X 0,Y 69.395,Z 1057.545,A -85,B 0,C 180,E1 -31601.686,E2 -31601.686} C_VEL
LIN {X 0,Y 65.802,Z 1058.101,A -85,B 0,C 180,E1 -31590,E2 -31590} C_VEL
LIN {X 0,Y 69.385,Z 1057.545,A -85,B 0,C 180,E1 -31578.312,E2 -31578.312} C_VEL
LIN {X 0,Y 75.767,Z 1056.055,A -85,B 0,C 180,E1 -31568.221,E2 -31568.221} C_VEL
LIN {X 0,Y 84.315,Z 1053.55,A -85,B 0,C 180,E1 -31559.993,E2 -31559.993} C_VEL
LIN {X 0,Y 96.935,Z 1048.97,A -85,B 0,C 180,E1 -31551.957,E2 -31551.957} C_VEL
LIN {X 0,Y 108.099,Z 1044.106,A -85,B 0,C 180,E1 -31546.95,E2 -31546.95} C_VEL
LIN {X 0,Y 119.922,Z 1038.123,A -85,B 0,C 180,E1 -31542.9,E2 -31542.9} C_VEL
LIN {X 0,Y 133.277,Z 1030.215,A -85,B 0,C 180,E1 -31539.362,E2 -31539.362} C_VEL
LIN {X 0,Y 146.522,Z 1020.954,A -85,B 0,C 180,E1 -31536.544,E2 -31536.544} C_VEL
LIN {X 0,Y 154.527,Z 1014.538,A -85,B 0,C 180,E1 -31535.052,E2 -31535.052} C_VEL
LIN {X 0,Y 155.366,Z 1014.496,A -85,B 0,C 180,E1 -31535.491,E2 -31535.491} C_VEL
LIN {X 0,Y 167.376,Z 1023.369,A -85,B 0,C 180,E1 -31547.793,E2 -31547.793} C_VEL
LIN {X 0,Y 179.27,Z 1029.094,A -85,B 0,C 180,E1 -31555.412,E2 -31555.412} C_VEL
LIN {X 0,Y 187.226,Z 1032.627,A -85,B 0,C 180,E1 -31559.694,E2 -31559.694} C_VEL
LIN {X 0,Y 197.083,Z 1036.951,A -85,B 0,C 180,E1 -31564.665,E2 -31564.665} C_VEL
LIN {X 0,Y 204.233,Z 1040.269,A -85,B 0,C 180,E1 -31568.295,E2 -31568.295} C_VEL
LIN {X 0,Y 208.61,Z 1042.439,A -85,B 0,C 180,E1 -31570.613,E2 -31570.613} C_VEL
LIN {X 0,Y 212.969,Z 1044.684,A -85,B 0,C 180,E1 -31573.134,E2 -31573.134} C_VEL
LIN {X 0,Y 217.282,Z 1047.124,A -85,B 0,C 180,E1 -31576.009,E2 -31576.009} C_VEL
LIN {X 0,Y 221.595,Z 1049.721,A -85,B 0,C 180,E1 -31579.471,E2 -31579.471} C_VEL
LIN {X 0,Y 225.063,Z 1051.6,A -85,B 0,C 180,E1 -31582.825,E2 -31582.825} C_VEL
LIN {X 0,Y 226.726,Z 1052.359,A -85,B 0,C 180,E1 -31584.664,E2 -31584.664} C_VEL
LIN {X 0,Y 227.895,Z 1052.806,A -85,B 0,C 180,E1 -31586.464,E2 -31586.464} C_VEL
LIN {X 0,Y 228.689,Z 1053.106,A -85,B 0,C 180,E1 -31588.239,E2 -31588.239} C_VEL
LIN {X 0,Y 229.021,Z 1053.215,A -85,B 0,C 180,E1 -31590,E2 -31590} C_VEL
LIN {X 0,Y 228.621,Z 1053.11,A -85,B 0,C 180,E1 -31591.762,E2 -31591.762} C_VEL
LIN {X 0,Y 227.835,Z 1052.811,A -85,B 0,C 180,E1 -31593.537,E2 -31593.537} C_VEL
LIN {X 0,Y 226.149,Z 1052.074,A -85,B 0,C 180,E1 -31596.043,E2 -31596.043} C_VEL
LIN {X 0,Y 223.183,Z 1050.583,A -85,B 0,C 180,E1 -31599.059,E2 -31599.059} C_VEL
LIN {X 0,Y 221.038,Z 1049.377,A -85,B 0,C 180,E1 -31600.998,E2 -31600.998} C_VEL
LIN {X 0,Y 217.285,Z 1047.121,A -85,B 0,C 180,E1 -31603.994,E2 -31603.994} C_VEL
LIN {X 0,Y 212.212,Z 1044.245,A -85,B 0,C 180,E1 -31607.341,E2 -31607.341} C_VEL
LIN {X 0,Y 207.961,Z 1042.08,A -85,B 0,C 180,E1 -31609.751,E2 -31609.751} C_VEL
LIN {X 0,Y 202.908,Z 1039.659,A -85,B 0,C 180,E1 -31612.395,E2 -31612.395} C_VEL
LIN {X 0,Y 196.397,Z 1036.648,A -85,B 0,C 180,E1 -31615.677,E2 -31615.677} C_VEL
LIN {X 0,Y 192.953,Z 1035.634,A -85,B 0,C 180,E1 -31617.051,E2 -31617.051} C_VEL
LIN {X 0,Y 185.84,Z 1034.71,A -85,B 0,C 180,E1 -31619.116,E2 -31619.116} C_VEL
LIN {X 0,Y 179.974,Z 1034.05,A -85,B 0,C 180,E1 -31620.815,E2 -31620.815} C_VEL
LIN {X 0,Y 176.141,Z 1033.236,A -85,B 0,C 180,E1 -31622.267,E2 -31622.267} C_VEL
LIN {X 0,Y 175.068,Z 1032.857,A -85,B 0,C 180,E1 -31622.8,E2 -31622.8} C_VEL
LIN {X 0,Y 163.214,Z 1027.68,A -85,B 0,C 180,E1 -31630.232,E2 -31630.232} C_VEL
LIN {X 0,Y 151.842,Z 1020.702,A -85,B 0,C 180,E1 -31640.83,E2 -31640.83} C_VEL
LIN {X 0,Y 149.302,Z 1021.935,A -85,B 0,C 180,E1 -31640.957,E2 -31640.957} C_VEL
LIN {X 0,Y 136.21,Z 1031.118,A -85,B 0,C 180,E1 -31637.876,E2 -31637.876} C_VEL
LIN {X 0,Y 124.931,Z 1037.918,A -85,B 0,C 180,E1 -31634.682,E2 -31634.682} C_VEL
LIN {X 0,Y 113.499,Z 1043.898,A -85,B 0,C 180,E1 -31630.553,E2 -31630.553} C_VEL
LIN {X 0,Y 102.72,Z 1048.764,A -85,B 0,C 180,E1 -31625.559,E2 -31625.559} C_VEL
LIN {X 0,Y 90.628,Z 1053.341,A -85,B 0,C 180,E1 -31617.728,E2 -31617.728} C_VEL
LIN {X 0,Y 81.767,Z 1056.033,A -85,B 0,C 180,E1 -31609.014,E2 -31609.014} C_VEL
LIN {X 0,Y 76.433,Z 1057.336,A -85,B 0,C 180,E1 -31600.597,E2 -31600.597} C_VEL
LIN {X 0,Y 72.972,Z 1057.893,A -85,B 0,C 180,E1 -31590,E2 -31590} C_VEL
LIN {X 0,Y 76.423,Z 1057.336,A -85,B 0,C 180,E1 -31579.402,E2 -31579.402} C_VEL
LIN {X 0,Y 82.495,Z 1055.845,A -85,B 0,C 180,E1 -31570.077,E2 -31570.077} C_VEL
LIN {X 0,Y 90.623,Z 1053.341,A -85,B 0,C 180,E1 -31562.27,E2 -31562.27} C_VEL
LIN {X 0,Y 102.719,Z 1048.764,A -85,B 0,C 180,E1 -31554.44,E2 -31554.44} C_VEL
LIN {X 0,Y 113.456,Z 1043.9,A -85,B 0,C 180,E1 -31549.428,E2 -31549.428} C_VEL
LIN {X 0,Y 124.927,Z 1037.918,A -85,B 0,C 180,E1 -31545.316,E2 -31545.316} C_VEL
LIN {X 0,Y 137.522,Z 1030.276,A -85,B 0,C 180,E1 -31541.776,E2 -31541.776} C_VEL
LIN {X 0,Y 149.335,Z 1021.933,A -85,B 0,C 180,E1 -31539.059,E2 -31539.059} C_VEL
LIN {X 0,Y 151.811,Z 1020.734,A -85,B 0,C 180,E1 -31539.184,E2 -31539.184} C_VEL
LIN {X 0,Y 164.156,Z 1028.11,A -85,B 0,C 180,E1 -31550.409,E2 -31550.409} C_VEL
LIN {X 0,Y 175.317,Z 1032.956,A -85,B 0,C 180,E1 -31557.333,E2 -31557.333} C_VEL
LIN {X 0,Y 186.106,Z 1037.307,A -85,B 0,C 180,E1 -31563.054,E2 -31563.054} C_VEL
LIN {X 0,Y 192.63,Z 1039.979,A -85,B 0,C 180,E1 -31566.339,E2 -31566.339} C_VEL
LIN {X 0,Y 198.299,Z 1042.376,A -85,B 0,C 180,E1 -31569.243,E2 -31569.243} C_VEL
LIN {X 0,Y 203.083,Z 1044.524,A -85,B 0,C 180,E1 -31571.853,E2 -31571.853} C_VEL
LIN {X 0,Y 207.126,Z 1046.451,A -85,B 0,C 180,E1 -31574.25,E2 -31574.25} C_VEL
LIN {X 0,Y 210.456,Z 1048.169,A -85,B 0,C 180,E1 -31576.482,E2 -31576.482} C_VEL
LIN {X 0,Y 214.361,Z 1050.245,A -85,B 0,C 180,E1 -31579.597,E2 -31579.597} C_VEL
LIN {X 0,Y 217.472,Z 1051.823,A -85,B 0,C 180,E1 -31582.573,E2 -31582.573} C_VEL
LIN {X 0,Y 219.37,Z 1052.607,A -85,B 0,C 180,E1 -31584.485,E2 -31584.485} C_VEL
LIN {X 0,Y 220.616,Z 1053.109,A -85,B 0,C 180,E1 -31586.347,E2 -31586.347} C_VEL
LIN {X 0,Y 221.514,Z 1053.434,A -85,B 0,C 180,E1 -31588.182,E2 -31588.182} C_VEL
LIN {X 0,Y 221.938,Z 1053.583,A -85,B 0,C 180,E1 -31590,E2 -31590} C_VEL
LIN {X 0,Y 221.447,Z 1053.436,A -85,B 0,C 180,E1 -31591.819,E2 -31591.819} C_VEL
LIN {X 0,Y 220.565,Z 1053.11,A -85,B 0,C 180,E1 -31593.654,E2 -31593.654} C_VEL
LIN {X 0,Y 219.015,Z 1052.458,A -85,B 0,C 180,E1 -31595.874,E2 -31595.874} C_VEL
LIN {X 0,Y 215.494,Z 1050.808,A -85,B 0,C 180,E1 -31599.385,E2 -31599.385} C_VEL
LIN {X 0,Y 213.121,Z 1049.611,A -85,B 0,C 180,E1 -31601.411,E2 -31601.411} C_VEL
LIN {X 0,Y 209.952,Z 1047.902,A -85,B 0,C 180,E1 -31603.894,E2 -31603.894} C_VEL
LIN {X 0,Y 205.529,Z 1045.662,A -85,B 0,C 180,E1 -31606.777,E2 -31606.777} C_VEL
LIN {X 0,Y 201.05,Z 1043.58,A -85,B 0,C 180,E1 -31609.299,E2 -31609.299} C_VEL
LIN {X 0,Y 196.595,Z 1041.602,A -85,B 0,C 180,E1 -31611.651,E2 -31611.651} C_VEL
LIN {X 0,Y 190.33,Z 1039.046,A -85,B 0,C 180,E1 -31614.79,E2 -31614.79} C_VEL
LIN {X 0,Y 183.537,Z 1036.26,A -85,B 0,C 180,E1 -31618.273,E2 -31618.273} C_VEL
LIN {X 0,Y 175.068,Z 1032.857,A -85,B 0,C 180,E1 -31622.8,E2 -31622.8} C_VEL
LIN {X 0,Y 171.607,Z 1031.941,A -85,B 0,C 180,E1 -31624.353,E2 -31624.353} C_VEL
LIN {X 0,Y 164.707,Z 1031.273,A -85,B 0,C 180,E1 -31626.771,E2 -31626.771} C_VEL
LIN {X 0,Y 159.243,Z 1030.83,A -85,B 0,C 180,E1 -31628.821,E2 -31628.821} C_VEL
LIN {X 0,Y 155.851,Z 1030.15,A -85,B 0,C 180,E1 -31630.576,E2 -31630.576} C_VEL
LIN {X 0,Y 154.959,Z 1029.805,A -85,B 0,C 180,E1 -31631.215,E2 -31631.215} C_VEL
LIN {X 0,Y 148.451,Z 1026.226,A -85,B 0,C 180,E1 -31637.206,E2 -31637.206} C_VEL
LIN {X 0,Y 146.755,Z 1027.061,A -85,B 0,C 180,E1 -31637.174,E2 -31637.174} C_VEL
LIN {X 0,Y 133.022,Z 1036.04,A -85,B 0,C 180,E1 -31633.379,E2 -31633.379} C_VEL
LIN {X 0,Y 121.768,Z 1042.342,A -85,B 0,C 180,E1 -31629.41,E2 -31629.41} C_VEL
LIN {X 0,Y 110.739,Z 1047.673,A -85,B 0,C 180,E1 -31624.41,E2 -31624.41} C_VEL
LIN {X 0,Y 101.501,Z 1051.478,A -85,B 0,C 180,E1 -31618.991,E2 -31618.991} C_VEL
LIN {X 0,Y 92.988,Z 1054.455,A -85,B 0,C 180,E1 -31612.203,E2 -31612.203} C_VEL
LIN {X 0,Y 86.134,Z 1056.459,A -85,B 0,C 180,E1 -31604.169,E2 -31604.169} C_VEL
LIN {X 0,Y 81.525,Z 1057.467,A -85,B 0,C 180,E1 -31594.945,E2 -31594.945} C_VEL
LIN {X 0,Y 80.132,Z 1057.686,A -85,B 0,C 180,E1 -31590,E2 -31590} C_VEL
LIN {X 0,Y 83.496,Z 1057.127,A -85,B 0,C 180,E1 -31580.309,E2 -31580.309} C_VEL
LIN {X 0,Y 89.297,Z 1055.636,A -85,B 0,C 180,E1 -31571.651,E2 -31571.651} C_VEL
LIN {X 0,Y 97.062,Z 1053.132,A -85,B 0,C 180,E1 -31564.251,E2 -31564.251} C_VEL
LIN {X 0,Y 108.527,Z 1048.618,A -85,B 0,C 180,E1 -31556.724,E2 -31556.724} C_VEL
LIN {X 0,Y 119.022,Z 1043.693,A -85,B 0,C 180,E1 -31551.685,E2 -31551.685} C_VEL
LIN {X 0,Y 130.13,Z 1037.714,A -85,B 0,C 180,E1 -31547.54,E2 -31547.54} C_VEL
LIN {X 0,Y 142.033,Z 1030.314,A -85,B 0,C 180,E1 -31544.034,E2 -31544.034} C_VEL
LIN {X 0,Y 146.776,Z 1027.048,A -85,B 0,C 180,E1 -31542.823,E2 -31542.823} C_VEL
LIN {X 0,Y 148.464,Z 1026.216,A -85,B 0,C 180,E1 -31542.79,E2 -31542.79} C_VEL
LIN {X 0,Y 159.807,Z 1031.936,A -85,B 0,C 180,E1 -31552.334,E2 -31552.334} C_VEL
LIN {X 0,Y 171.439,Z 1036.525,A -85,B 0,C 180,E1 -31559.413,E2 -31559.413} C_VEL
LIN {X 0,Y 181.838,Z 1040.319,A -85,B 0,C 180,E1 -31564.841,E2 -31564.841} C_VEL
LIN {X 0,Y 188.901,Z 1042.993,A -85,B 0,C 180,E1 -31568.451,E2 -31568.451} C_VEL
LIN {X 0,Y 193.609,Z 1044.814,A -85,B 0,C 180,E1 -31570.932,E2 -31570.932} C_VEL
LIN {X 0,Y 198.238,Z 1046.72,A -85,B 0,C 180,E1 -31573.524,E2 -31573.524} C_VEL
LIN {X 0,Y 202.57,Z 1048.647,A -85,B 0,C 180,E1 -31576.269,E2 -31576.269} C_VEL
LIN {X 0,Y 207.114,Z 1050.767,A -85,B 0,C 180,E1 -31579.75,E2 -31579.75} C_VEL
LIN {X 0,Y 209.863,Z 1052.046,A -85,B 0,C 180,E1 -31582.302,E2 -31582.302} C_VEL
LIN {X 0,Y 211.879,Z 1052.835,A -85,B 0,C 180,E1 -31584.313,E2 -31584.313} C_VEL
LIN {X 0,Y 213.329,Z 1053.322,A -85,B 0,C 180,E1 -31586.222,E2 -31586.222} C_VEL
LIN {X 0,Y 214.315,Z 1053.643,A -85,B 0,C 180,E1 -31588.121,E2 -31588.121} C_VEL
LIN {X 0,Y 214.831,Z 1053.788,A -85,B 0,C 180,E1 -31590,E2 -31590} C_VEL
LIN {X 0,Y 214.251,Z 1053.644,A -85,B 0,C 180,E1 -31591.88,E2 -31591.88} C_VEL
LIN {X 0,Y 213.289,Z 1053.323,A -85,B 0,C 180,E1 -31593.779,E2 -31593.779} C_VEL
LIN {X 0,Y 211.845,Z 1052.826,A -85,B 0,C 180,E1 -31595.712,E2 -31595.712} C_VEL
LIN {X 0,Y 209.864,Z 1052.047,A -85,B 0,C 180,E1 -31597.698,E2 -31597.698} C_VEL
LIN {X 0,Y 207.116,Z 1050.765,A -85,B 0,C 180,E1 -31600.253,E2 -31600.253} C_VEL
LIN {X 0,Y 202.573,Z 1048.644,A -85,B 0,C 180,E1 -31603.734,E2 -31603.734} C_VEL
LIN {X 0,Y 198.031,Z 1046.612,A -85,B 0,C 180,E1 -31606.625,E2 -31606.625} C_VEL
LIN {X 0,Y 193.462,Z 1044.723,A -85,B 0,C 180,E1 -31609.179,E2 -31609.179} C_VEL
LIN {X 0,Y 188.138,Z 1042.69,A -85,B 0,C 180,E1 -31611.934,E2 -31611.934} C_VEL
LIN {X 0,Y 179.991,Z 1039.658,A -85,B 0,C 180,E1 -31616.097,E2 -31616.097} C_VEL
LIN {X 0,Y 171.451,Z 1036.514,A -85,B 0,C 180,E1 -31620.593,E2 -31620.593} C_VEL
LIN {X 0,Y 159.782,Z 1031.958,A -85,B 0,C 180,E1 -31627.654,E2 -31627.654} C_VEL
LIN {X 0,Y 154.959,Z 1029.805,A -85,B 0,C 180,E1 -31631.215,E2 -31631.215} C_VEL
LIN {X 0,Y 153.321,Z 1029.766,A -85,B 0,C 180,E1 -31631.86,E2 -31631.86} C_VEL
